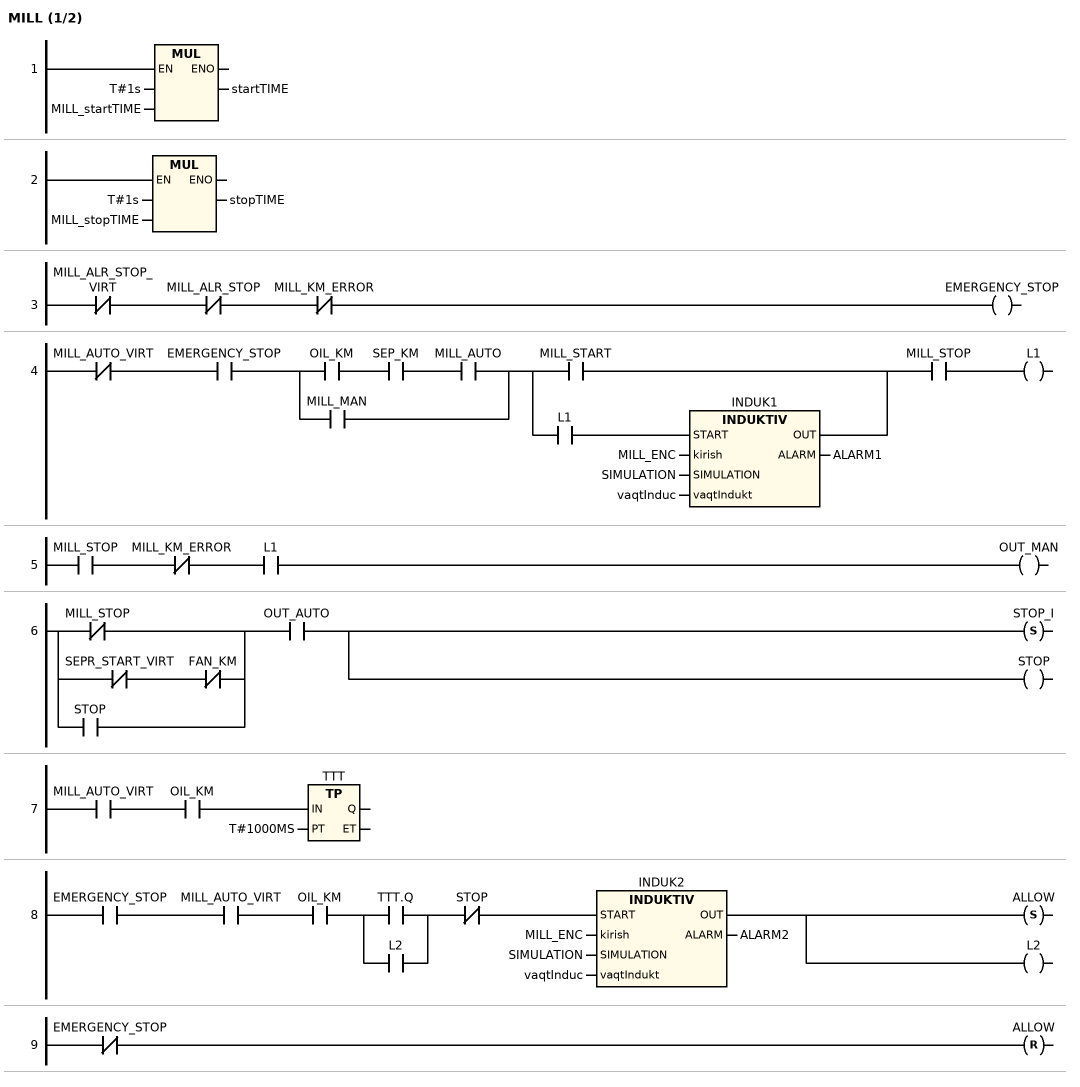
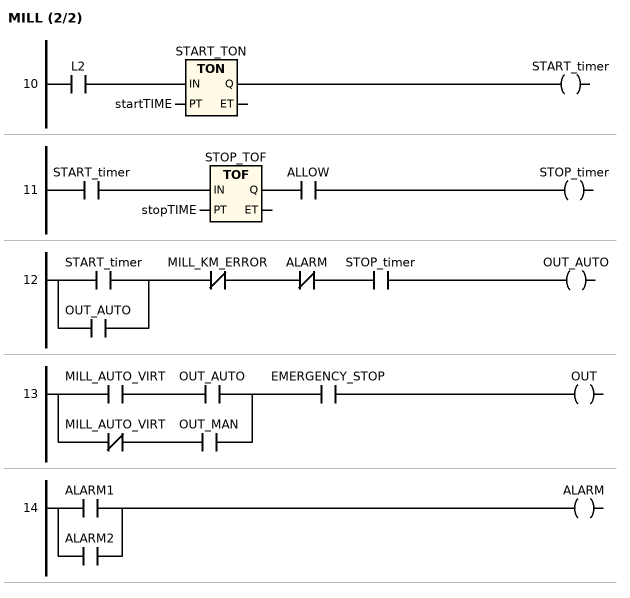
_LD_ (* Ladder Diagram *)
NETWORK 1
	*
		EN --- MUL(T#1s, MILL_startTIME) => startTIME
NETWORK 2
	*
		EN --- MUL(T#1s, MILL_stopTIME) => stopTIME
NETWORK 3
	[/MILL_ALR_STOP_VIRT] - [/MILL_ALR_STOP] - [/MILL_KM_ERROR] --- (EMERGENCY_STOP)
NETWORK 4
	[/MILL_AUTO_VIRT] - [EMERGENCY_STOP] - { [OIL_KM] - [SEP_KM] - [MILL_AUTO] | [MILL_MAN] } - { [MILL_START] | [L1] - INDUK1:INDUKTIV(START: *, kirish: MILL_ENC, SIMULATION: SIMULATION, vaqtIndukt: vaqtInduc, ALARM => ALARM1) } - [MILL_STOP] --- (L1)
NETWORK 5
	[MILL_STOP] - [/MILL_KM_ERROR] - [L1] --- (OUT_MAN)
NETWORK 6
	{ [/MILL_STOP] | [/SEPR_START_VIRT] - [/FAN_KM] | [STOP] } - [OUT_AUTO] --- (S STOP_I) (STOP)
NETWORK 7
	[MILL_AUTO_VIRT] - [OIL_KM] - TTT:TP(IN: *, PT: T#1000MS)
NETWORK 8
	[EMERGENCY_STOP] - [MILL_AUTO_VIRT] - [OIL_KM] - { [TTT.Q] | [L2] } - [/STOP] - INDUK2:INDUKTIV(START: *, kirish: MILL_ENC, SIMULATION: SIMULATION, vaqtIndukt: vaqtInduc, ALARM => ALARM2) --- (S ALLOW) (L2)
NETWORK 9
	[/EMERGENCY_STOP] --- (R ALLOW)
NETWORK 10
	[L2] - START_TON:TON(IN: *, PT: startTIME) --- (START_timer)
NETWORK 11
	[START_timer] - STOP_TOF:TOF(IN: *, PT: stopTIME) - [ALLOW] --- (STOP_timer)
NETWORK 12
	{ [START_timer] | [OUT_AUTO] } - [/MILL_KM_ERROR] - [/ALARM] - [STOP_timer] --- (OUT_AUTO)
NETWORK 13
	{ [MILL_AUTO_VIRT] - [OUT_AUTO] | [/MILL_AUTO_VIRT] - [OUT_MAN] } - [EMERGENCY_STOP] --- (OUT)
NETWORK 14
	{ [ALARM1] | [ALARM2] } --- (ALARM)
_END_LD_
(* the same logic as Structured Text *)
(* Network 1 *)
startTIME := T#1s * MILL_startTIME;
(* Network 2 *)
stopTIME := T#1s * MILL_stopTIME;
(* Network 3 *)
EMERGENCY_STOP := NOT MILL_ALR_STOP_VIRT AND NOT MILL_ALR_STOP AND NOT MILL_KM_ERROR;
(* Network 4 *)
_p1 := NOT MILL_AUTO_VIRT AND EMERGENCY_STOP AND (OIL_KM AND SEP_KM AND MILL_AUTO OR MILL_MAN);
INDUK1(START := _p1 AND L1, kirish := MILL_ENC, SIMULATION := SIMULATION, vaqtIndukt := vaqtInduc);
ALARM1 := INDUK1.ALARM;
L1 := (_p1 AND MILL_START OR INDUK1.OUT) AND MILL_STOP;
(* Network 5 *)
OUT_MAN := MILL_STOP AND NOT MILL_KM_ERROR AND L1;
(* Network 6 *)
_p2 := (NOT MILL_STOP OR NOT SEPR_START_VIRT AND NOT FAN_KM OR STOP) AND OUT_AUTO;
IF _p2 THEN STOP_I := TRUE; END_IF;
STOP := _p2;
(* Network 7 *)
TTT(IN := MILL_AUTO_VIRT AND OIL_KM, PT := T#1000MS);
(* Network 8 *)
INDUK2(START := EMERGENCY_STOP AND MILL_AUTO_VIRT AND OIL_KM AND (TTT.Q OR L2) AND NOT STOP, kirish := MILL_ENC, SIMULATION := SIMULATION, vaqtIndukt := vaqtInduc);
ALARM2 := INDUK2.ALARM;
IF INDUK2.OUT THEN ALLOW := TRUE; END_IF;
L2 := INDUK2.OUT;
(* Network 9 *)
IF NOT EMERGENCY_STOP THEN ALLOW := FALSE; END_IF;
(* Network 10 *)
START_TON(IN := L2, PT := startTIME);
START_timer := START_TON.Q;
(* Network 11 *)
STOP_TOF(IN := START_timer, PT := stopTIME);
STOP_timer := STOP_TOF.Q AND ALLOW;
(* Network 12 *)
OUT_AUTO := (START_timer OR OUT_AUTO) AND NOT MILL_KM_ERROR AND NOT ALARM AND STOP_timer;
(* Network 13 *)
OUT := (MILL_AUTO_VIRT AND OUT_AUTO OR NOT MILL_AUTO_VIRT AND OUT_MAN) AND EMERGENCY_STOP;
(* Network 14 *)
ALARM := ALARM1 OR ALARM2;
END_FUNCTION_BLOCK

(* POU FAN, LD *)
FUNCTION_BLOCK FAN
VAR_INPUT
	EN : BOOL;
	MILL_ALR_STOP: BOOL;
	MILL_ALR_STOP_VIRT : BOOL;
	MILL_AUTO : BOOL;
	MILL_AUTO_VIRT : BOOL;
	MILL_MAN : BOOL;
	FAN_START : BOOL;
	VIBRATOR_T : BOOL;

	FAN_STOP : BOOL;
	MILL_KM : BOOL;

	FAN_KM_ERROR : BOOL;
	SEPR_START_VIRT : BOOL;
	FAN_startTIME : WORD;
	FAN_stopTIME : WORD;
END_VAR

VAR_OUTPUT
	OUT : BOOL;
	ALARM : BOOL;
END_VAR
VAR
	INDUK1: INDUKTIV;
	INDUK2: INDUKTIV;
	OUT_MAN: BOOL;
	OUT_AUTO: BOOL;
	START_TON : TON;
	STOP_TOF : TOF;
	startTIME : TIME;
	stopTIME : TIME;
	L1: BOOL;
	L2: BOOL;
	ES: BOOL;
	EMERGENCY_STOP: BOOL;
	ALARM1 : BOOL;
	ALARM2 : BOOL;

	STOP: BOOL;
	ALLOW: BOOL;
	START_timer: BOOL;
	STOP_timer: BOOL;
	TTT : TP;
END_VAR
VAR (* helpers for the ST form of the networks *)
	_p1 : BOOL;
END_VAR
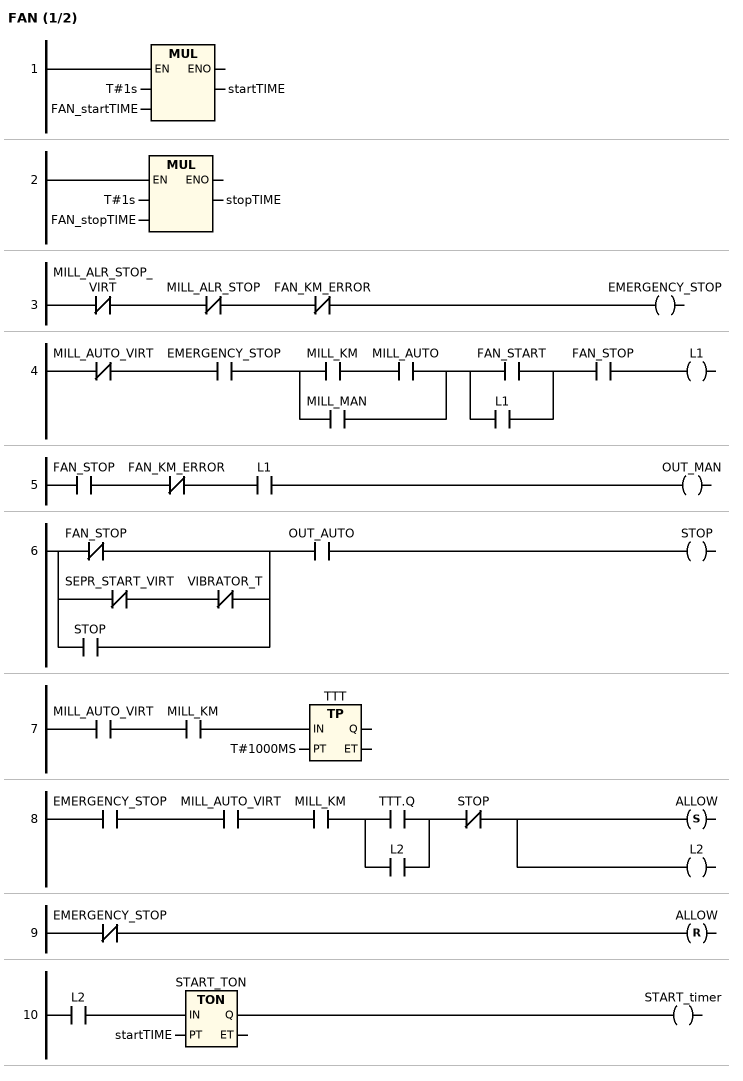
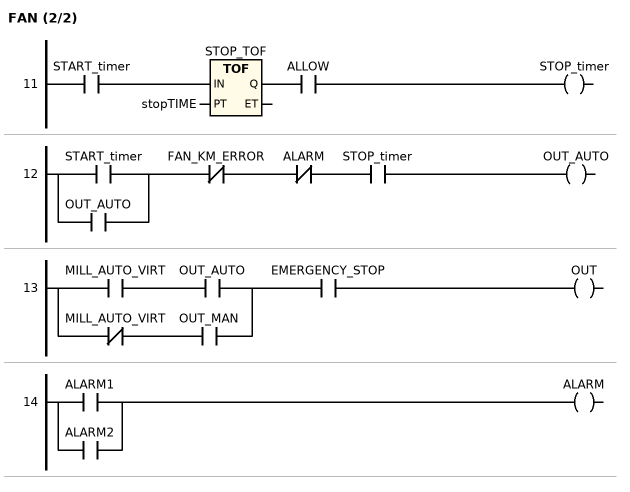
_LD_ (* Ladder Diagram *)
NETWORK 1
	*
		EN --- MUL(T#1s, FAN_startTIME) => startTIME
NETWORK 2
	*
		EN --- MUL(T#1s, FAN_stopTIME) => stopTIME
NETWORK 3
	[/MILL_ALR_STOP_VIRT] - [/MILL_ALR_STOP] - [/FAN_KM_ERROR] --- (EMERGENCY_STOP)
NETWORK 4
	[/MILL_AUTO_VIRT] - [EMERGENCY_STOP] - { [MILL_KM] - [MILL_AUTO] | [MILL_MAN] } - { [FAN_START] | [L1] } - [FAN_STOP] --- (L1)
NETWORK 5
	[FAN_STOP] - [/FAN_KM_ERROR] - [L1] --- (OUT_MAN)
NETWORK 6
	{ [/FAN_STOP] | [/SEPR_START_VIRT] - [/VIBRATOR_T] | [STOP] } - [OUT_AUTO] --- (STOP)
NETWORK 7
	[MILL_AUTO_VIRT] - [MILL_KM] - TTT:TP(IN: *, PT: T#1000MS)
NETWORK 8
	[EMERGENCY_STOP] - [MILL_AUTO_VIRT] - [MILL_KM] - { [TTT.Q] | [L2] } - [/STOP] --- (S ALLOW) (L2)
NETWORK 9
	[/EMERGENCY_STOP] --- (R ALLOW)
NETWORK 10
	[L2] - START_TON:TON(IN: *, PT: startTIME) --- (START_timer)
NETWORK 11
	[START_timer] - STOP_TOF:TOF(IN: *, PT: stopTIME) - [ALLOW] --- (STOP_timer)
NETWORK 12
	{ [START_timer] | [OUT_AUTO] } - [/FAN_KM_ERROR] - [/ALARM] - [STOP_timer] --- (OUT_AUTO)
NETWORK 13
	{ [MILL_AUTO_VIRT] - [OUT_AUTO] | [/MILL_AUTO_VIRT] - [OUT_MAN] } - [EMERGENCY_STOP] --- (OUT)
NETWORK 14
	{ [ALARM1] | [ALARM2] } --- (ALARM)
_END_LD_
(* the same logic as Structured Text *)
(* Network 1 *)
startTIME := T#1s * FAN_startTIME;
(* Network 2 *)
stopTIME := T#1s * FAN_stopTIME;
(* Network 3 *)
EMERGENCY_STOP := NOT MILL_ALR_STOP_VIRT AND NOT MILL_ALR_STOP AND NOT FAN_KM_ERROR;
(* Network 4 *)
L1 := NOT MILL_AUTO_VIRT AND EMERGENCY_STOP AND (MILL_KM AND MILL_AUTO OR MILL_MAN) AND (FAN_START OR L1) AND FAN_STOP;
(* Network 5 *)
OUT_MAN := FAN_STOP AND NOT FAN_KM_ERROR AND L1;
(* Network 6 *)
STOP := (NOT FAN_STOP OR NOT SEPR_START_VIRT AND NOT VIBRATOR_T OR STOP) AND OUT_AUTO;
(* Network 7 *)
TTT(IN := MILL_AUTO_VIRT AND MILL_KM, PT := T#1000MS);
(* Network 8 *)
_p1 := EMERGENCY_STOP AND MILL_AUTO_VIRT AND MILL_KM AND (TTT.Q OR L2) AND NOT STOP;
IF _p1 THEN ALLOW := TRUE; END_IF;
L2 := _p1;
(* Network 9 *)
IF NOT EMERGENCY_STOP THEN ALLOW := FALSE; END_IF;
(* Network 10 *)
START_TON(IN := L2, PT := startTIME);
START_timer := START_TON.Q;
(* Network 11 *)
STOP_TOF(IN := START_timer, PT := stopTIME);
STOP_timer := STOP_TOF.Q AND ALLOW;
(* Network 12 *)
OUT_AUTO := (START_timer OR OUT_AUTO) AND NOT FAN_KM_ERROR AND NOT ALARM AND STOP_timer;
(* Network 13 *)
OUT := (MILL_AUTO_VIRT AND OUT_AUTO OR NOT MILL_AUTO_VIRT AND OUT_MAN) AND EMERGENCY_STOP;
(* Network 14 *)
ALARM := ALARM1 OR ALARM2;
END_FUNCTION_BLOCK

(* POU CONV, LD *)
FUNCTION_BLOCK CONV
VAR_INPUT
	EN : BOOL;
	MILL_ALR_STOP: BOOL;
	MILL_ALR_STOP_VIRT : BOOL;
	MILL_AUTO : BOOL;
	MILL_AUTO_VIRT : BOOL;
	MILL_MAN : BOOL;
	CONV_START : BOOL;
	FAN_KM : BOOL;
	MILL_KM : BOOL;
	CONV_ENC : BOOL;
	CONV_STOP : BOOL;
	VIBRATOR_T : BOOL;
	CONV_KM_ERROR : BOOL;
	SIMULATION : BOOL := TRUE;
	MATER_FULL : BOOL;
	SEPR_START_VIRT : BOOL;
	vaqtInduc : WORD := 15;
END_VAR

VAR_OUTPUT
	OUT : BOOL;
	ALARM : BOOL;
END_VAR
VAR
	INDUK1: INDUKTIV;
	INDUK2: INDUKTIV;
	OUT_MAN: BOOL;
	OUT_AUTO: BOOL;
	START_TON : TON;
	STOP_TOF : TOF;
	startTIME : TIME;
	stopTIME : TIME;
	L1: BOOL;
	L2: BOOL;
	ES: BOOL;
	EMERGENCY_STOP: BOOL;
	ALARM1 : BOOL;
	ALARM2 : BOOL;

	STOP: BOOL;
	ALLOW: BOOL;
	START_timer: BOOL;
	STOP_timer: BOOL;
	TTT : TP;
END_VAR
VAR (* helpers for the ST form of the networks *)
	_p1 : BOOL;
END_VAR
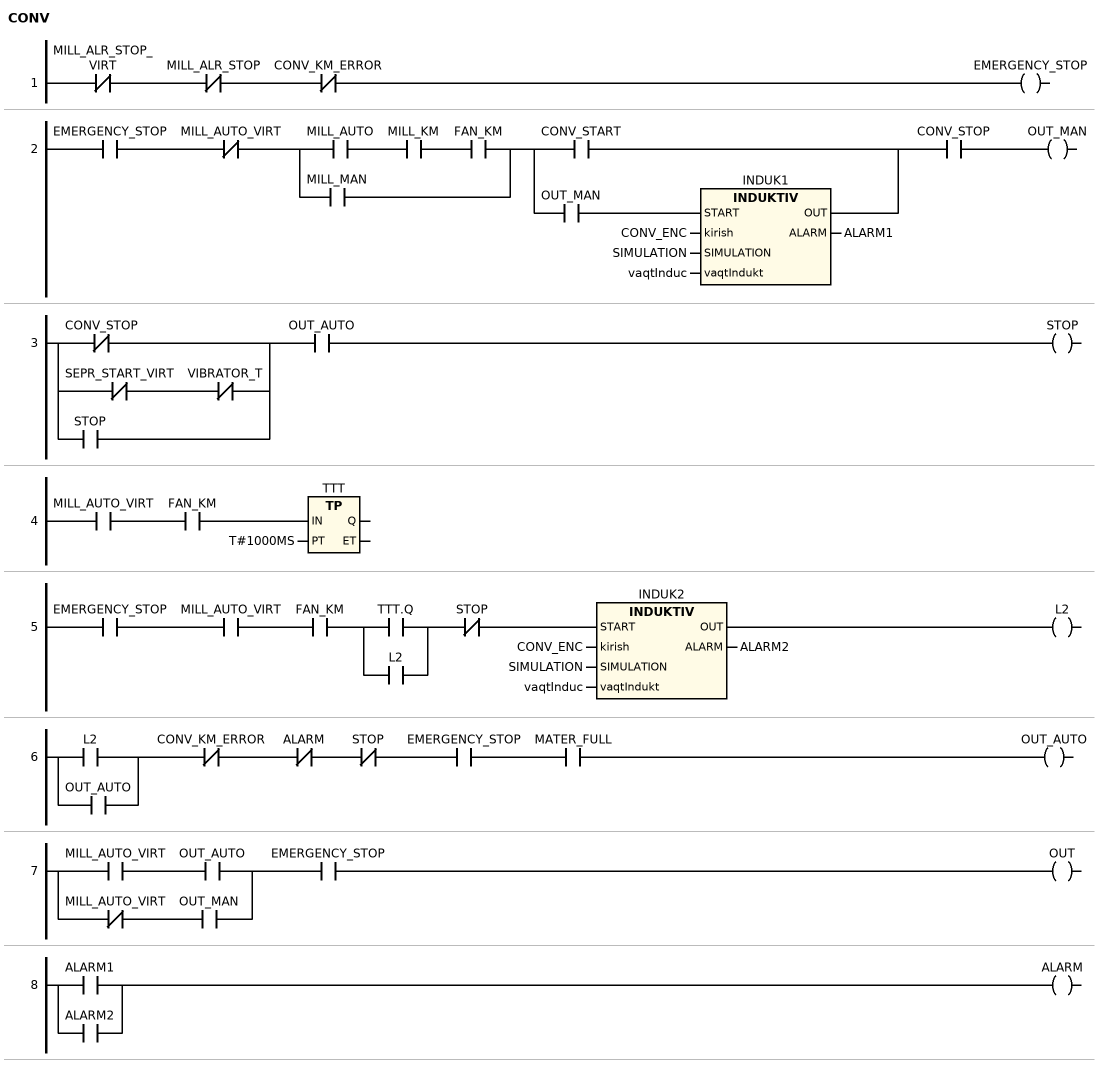
_LD_ (* Ladder Diagram *)
NETWORK 1
	[/MILL_ALR_STOP_VIRT] - [/MILL_ALR_STOP] - [/CONV_KM_ERROR] --- (EMERGENCY_STOP)
NETWORK 2
	[EMERGENCY_STOP] - [/MILL_AUTO_VIRT] - { [MILL_AUTO] - [MILL_KM] - [FAN_KM] | [MILL_MAN] } - { [CONV_START] | [OUT_MAN] - INDUK1:INDUKTIV(START: *, kirish: CONV_ENC, SIMULATION: SIMULATION, vaqtIndukt: vaqtInduc, ALARM => ALARM1) } - [CONV_STOP] --- (OUT_MAN)
NETWORK 3
	{ [/CONV_STOP] | [/SEPR_START_VIRT] - [/VIBRATOR_T] | [STOP] } - [OUT_AUTO] --- (STOP)
NETWORK 4
	[MILL_AUTO_VIRT] - [FAN_KM] - TTT:TP(IN: *, PT: T#1000MS)
NETWORK 5
	[EMERGENCY_STOP] - [MILL_AUTO_VIRT] - [FAN_KM] - { [TTT.Q] | [L2] } - [/STOP] - INDUK2:INDUKTIV(START: *, kirish: CONV_ENC, SIMULATION: SIMULATION, vaqtIndukt: vaqtInduc, ALARM => ALARM2) --- (L2)
NETWORK 6
	{ [L2] | [OUT_AUTO] } - [/CONV_KM_ERROR] - [/ALARM] - [/STOP] - [EMERGENCY_STOP] - [MATER_FULL] --- (OUT_AUTO)
NETWORK 7
	{ [MILL_AUTO_VIRT] - [OUT_AUTO] | [/MILL_AUTO_VIRT] - [OUT_MAN] } - [EMERGENCY_STOP] --- (OUT)
NETWORK 8
	{ [ALARM1] | [ALARM2] } --- (ALARM)
_END_LD_
(* the same logic as Structured Text *)
(* Network 1 *)
EMERGENCY_STOP := NOT MILL_ALR_STOP_VIRT AND NOT MILL_ALR_STOP AND NOT CONV_KM_ERROR;
(* Network 2 *)
_p1 := EMERGENCY_STOP AND NOT MILL_AUTO_VIRT AND (MILL_AUTO AND MILL_KM AND FAN_KM OR MILL_MAN);
INDUK1(START := _p1 AND OUT_MAN, kirish := CONV_ENC, SIMULATION := SIMULATION, vaqtIndukt := vaqtInduc);
ALARM1 := INDUK1.ALARM;
OUT_MAN := (_p1 AND CONV_START OR INDUK1.OUT) AND CONV_STOP;
(* Network 3 *)
STOP := (NOT CONV_STOP OR NOT SEPR_START_VIRT AND NOT VIBRATOR_T OR STOP) AND OUT_AUTO;
(* Network 4 *)
TTT(IN := MILL_AUTO_VIRT AND FAN_KM, PT := T#1000MS);
(* Network 5 *)
INDUK2(START := EMERGENCY_STOP AND MILL_AUTO_VIRT AND FAN_KM AND (TTT.Q OR L2) AND NOT STOP, kirish := CONV_ENC, SIMULATION := SIMULATION, vaqtIndukt := vaqtInduc);
ALARM2 := INDUK2.ALARM;
L2 := INDUK2.OUT;
(* Network 6 *)
OUT_AUTO := (L2 OR OUT_AUTO) AND NOT CONV_KM_ERROR AND NOT ALARM AND NOT STOP AND EMERGENCY_STOP AND MATER_FULL;
(* Network 7 *)
OUT := (MILL_AUTO_VIRT AND OUT_AUTO OR NOT MILL_AUTO_VIRT AND OUT_MAN) AND EMERGENCY_STOP;
(* Network 8 *)
ALARM := ALARM1 OR ALARM2;
END_FUNCTION_BLOCK

(* POU ALARMS, LD *)
PROGRAM ALARMS
VAR
	tofELV: TON;
	tofSHNK3: TON;
	tofSHNK4: TON;
	tofSHNK_SKL_3: TON;
	tofSHNK_SKL_4: TON;
	tofSTAR_31: TON;
	tofSTAR_32: TON;
	tofSTAR_41: TON;
	tofSTAR_42: TON;
	tofSEPR_3: TON;
	tofSEPR_4: TON;
	tofOIL_3: TON;
	tofOIL_4: TON;
	tofMILL_3: TON;
	tofMILL_4: TON;
	tofFAN_3: TON;
	tofFAN_4: TON;
	tofCONV_3: TON;
	tofCONV_4: TON;
	tofVIB_3: TON;
	tofVIB_4: TON;

	vaqt : TIME := T#30S;
END_VAR
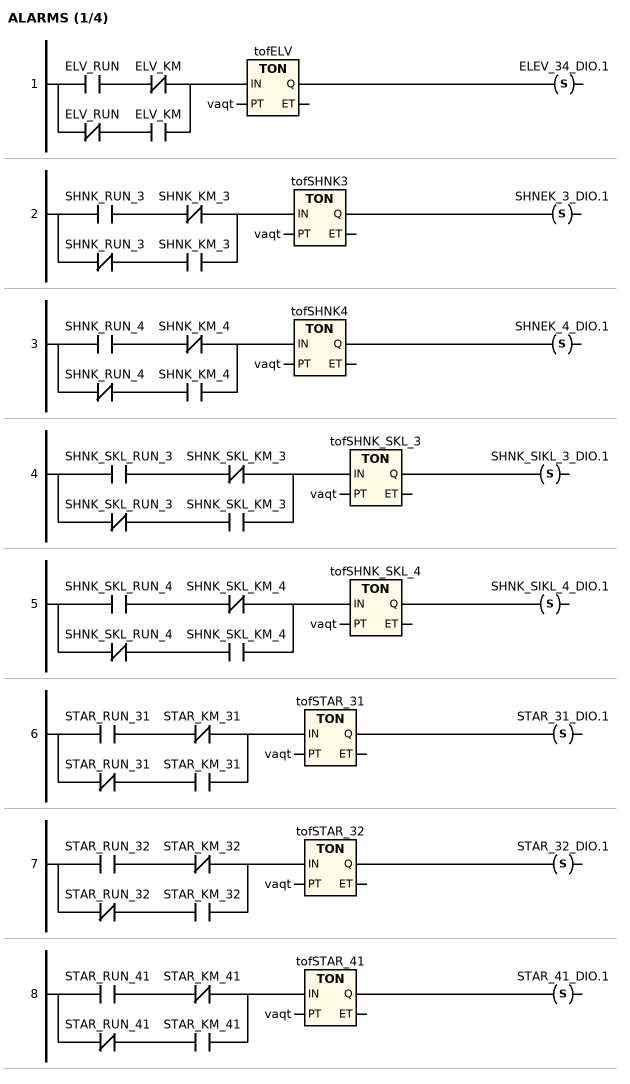
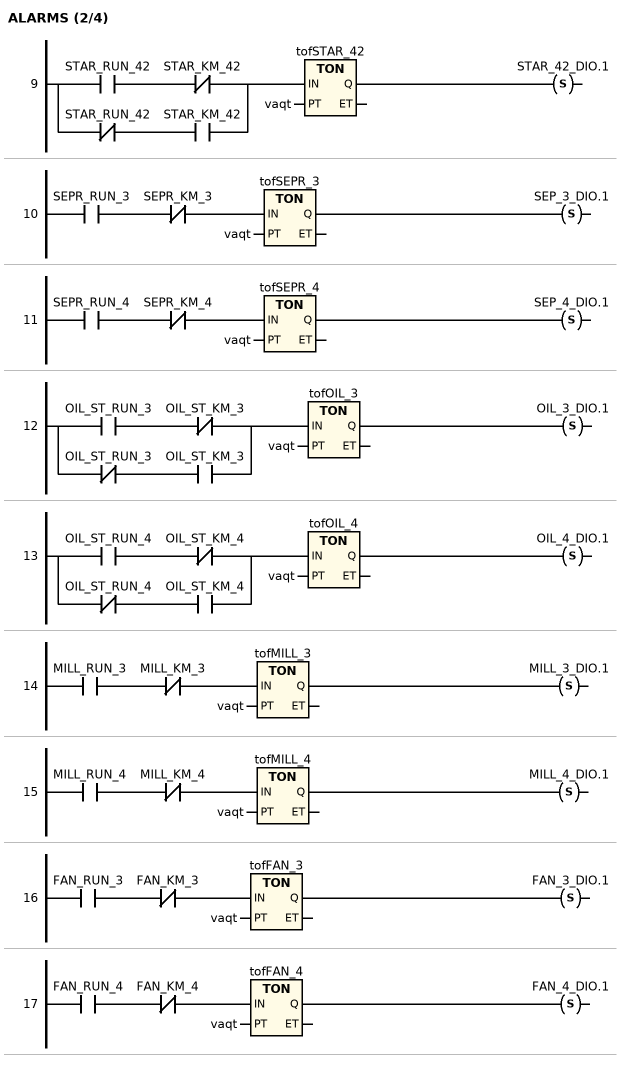
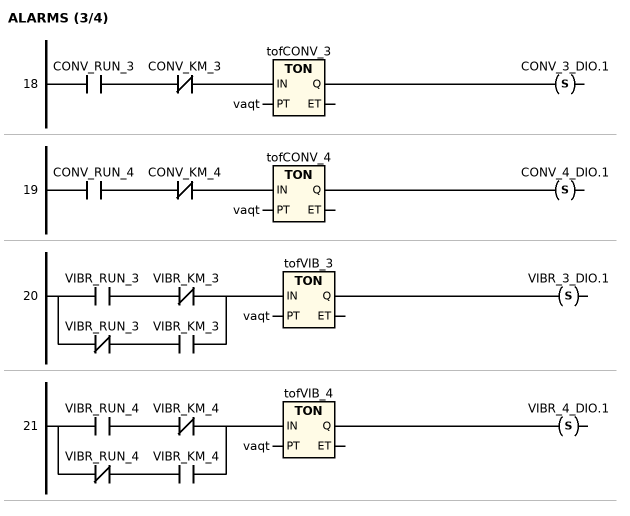
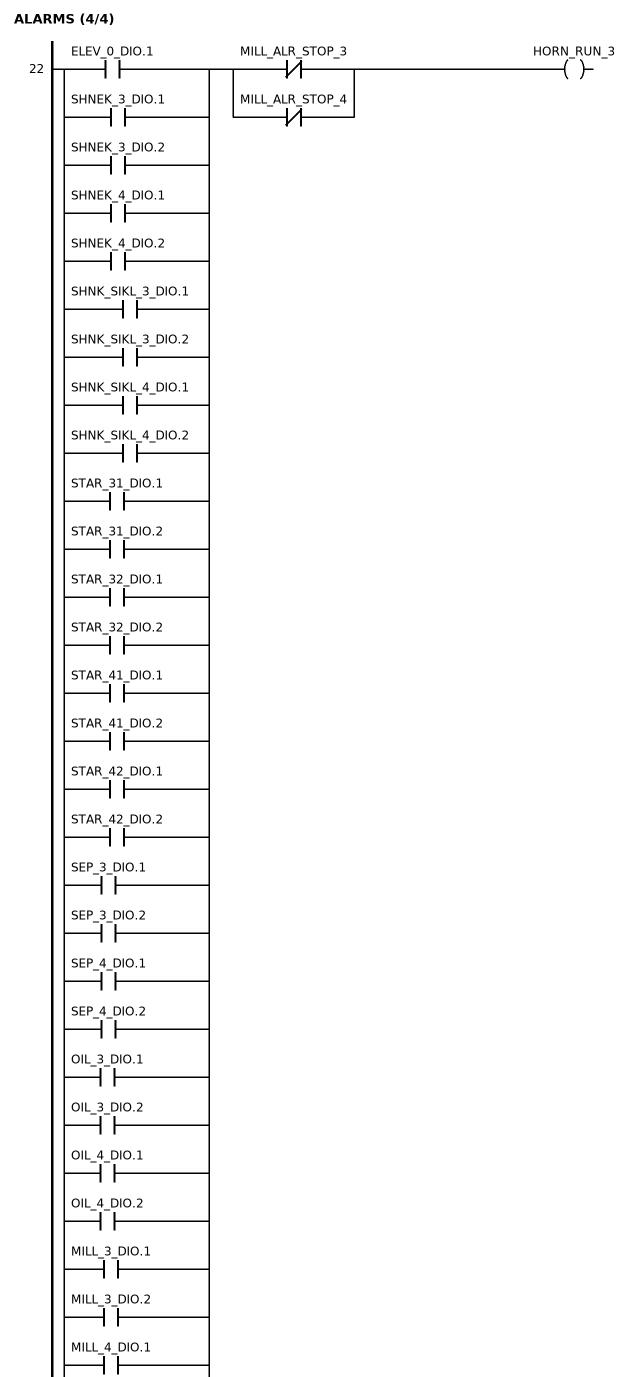
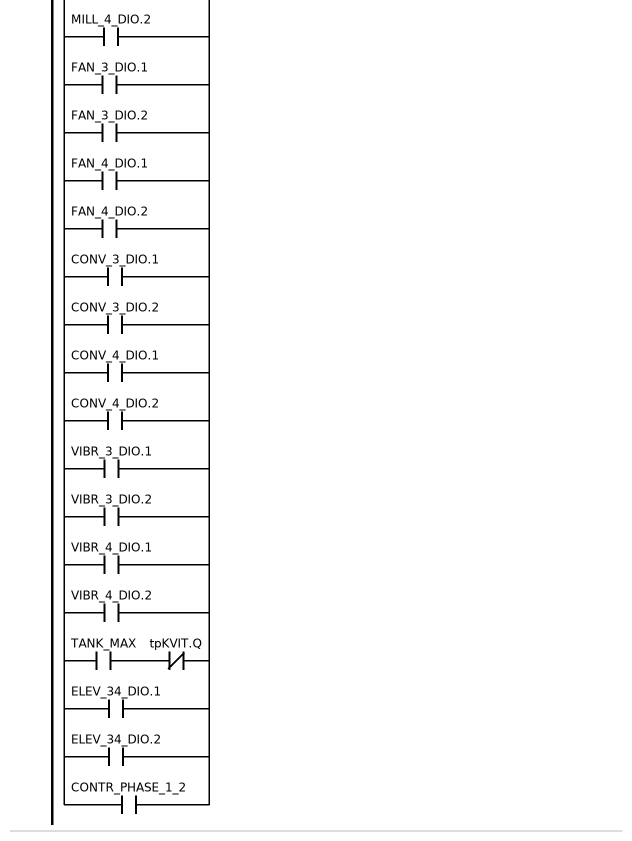
_LD_ (* Ladder Diagram *)
NETWORK 1
	{ [ELV_RUN] - [/ELV_KM] | [/ELV_RUN] - [ELV_KM] } - tofELV:TON(IN: *, PT: vaqt) --- (S ELEV_34_DIO.1)
NETWORK 2
	{ [SHNK_RUN_3] - [/SHNK_KM_3] | [/SHNK_RUN_3] - [SHNK_KM_3] } - tofSHNK3:TON(IN: *, PT: vaqt) --- (S SHNEK_3_DIO.1)
NETWORK 3
	{ [SHNK_RUN_4] - [/SHNK_KM_4] | [/SHNK_RUN_4] - [SHNK_KM_4] } - tofSHNK4:TON(IN: *, PT: vaqt) --- (S SHNEK_4_DIO.1)
NETWORK 4
	{ [SHNK_SKL_RUN_3] - [/SHNK_SKL_KM_3] | [/SHNK_SKL_RUN_3] - [SHNK_SKL_KM_3] } - tofSHNK_SKL_3:TON(IN: *, PT: vaqt) --- (S SHNK_SIKL_3_DIO.1)
NETWORK 5
	{ [SHNK_SKL_RUN_4] - [/SHNK_SKL_KM_4] | [/SHNK_SKL_RUN_4] - [SHNK_SKL_KM_4] } - tofSHNK_SKL_4:TON(IN: *, PT: vaqt) --- (S SHNK_SIKL_4_DIO.1)
NETWORK 6
	{ [STAR_RUN_31] - [/STAR_KM_31] | [/STAR_RUN_31] - [STAR_KM_31] } - tofSTAR_31:TON(IN: *, PT: vaqt) --- (S STAR_31_DIO.1)
NETWORK 7
	{ [STAR_RUN_32] - [/STAR_KM_32] | [/STAR_RUN_32] - [STAR_KM_32] } - tofSTAR_32:TON(IN: *, PT: vaqt) --- (S STAR_32_DIO.1)
NETWORK 8
	{ [STAR_RUN_41] - [/STAR_KM_41] | [/STAR_RUN_41] - [STAR_KM_41] } - tofSTAR_41:TON(IN: *, PT: vaqt) --- (S STAR_41_DIO.1)
NETWORK 9
	{ [STAR_RUN_42] - [/STAR_KM_42] | [/STAR_RUN_42] - [STAR_KM_42] } - tofSTAR_42:TON(IN: *, PT: vaqt) --- (S STAR_42_DIO.1)
NETWORK 10
	[SEPR_RUN_3] - [/SEPR_KM_3] - tofSEPR_3:TON(IN: *, PT: vaqt) --- (S SEP_3_DIO.1)
NETWORK 11
	[SEPR_RUN_4] - [/SEPR_KM_4] - tofSEPR_4:TON(IN: *, PT: vaqt) --- (S SEP_4_DIO.1)
NETWORK 12
	{ [OIL_ST_RUN_3] - [/OIL_ST_KM_3] | [/OIL_ST_RUN_3] - [OIL_ST_KM_3] } - tofOIL_3:TON(IN: *, PT: vaqt) --- (S OIL_3_DIO.1)
NETWORK 13
	{ [OIL_ST_RUN_4] - [/OIL_ST_KM_4] | [/OIL_ST_RUN_4] - [OIL_ST_KM_4] } - tofOIL_4:TON(IN: *, PT: vaqt) --- (S OIL_4_DIO.1)
NETWORK 14
	[MILL_RUN_3] - [/MILL_KM_3] - tofMILL_3:TON(IN: *, PT: vaqt) --- (S MILL_3_DIO.1)
NETWORK 15
	[MILL_RUN_4] - [/MILL_KM_4] - tofMILL_4:TON(IN: *, PT: vaqt) --- (S MILL_4_DIO.1)
NETWORK 16
	[FAN_RUN_3] - [/FAN_KM_3] - tofFAN_3:TON(IN: *, PT: vaqt) --- (S FAN_3_DIO.1)
NETWORK 17
	[FAN_RUN_4] - [/FAN_KM_4] - tofFAN_4:TON(IN: *, PT: vaqt) --- (S FAN_4_DIO.1)
NETWORK 18
	[CONV_RUN_3] - [/CONV_KM_3] - tofCONV_3:TON(IN: *, PT: vaqt) --- (S CONV_3_DIO.1)
NETWORK 19
	[CONV_RUN_4] - [/CONV_KM_4] - tofCONV_4:TON(IN: *, PT: vaqt) --- (S CONV_4_DIO.1)
NETWORK 20
	{ [VIBR_RUN_3] - [/VIBR_KM_3] | [/VIBR_RUN_3] - [VIBR_KM_3] } - tofVIB_3:TON(IN: *, PT: vaqt) --- (S VIBR_3_DIO.1)
NETWORK 21
	{ [VIBR_RUN_4] - [/VIBR_KM_4] | [/VIBR_RUN_4] - [VIBR_KM_4] } - tofVIB_4:TON(IN: *, PT: vaqt) --- (S VIBR_4_DIO.1)
NETWORK 22
	{ [ELEV_0_DIO.1] | [SHNEK_3_DIO.1] | [SHNEK_3_DIO.2] | [SHNEK_4_DIO.1] | [SHNEK_4_DIO.2] | [SHNK_SIKL_3_DIO.1] | [SHNK_SIKL_3_DIO.2] | [SHNK_SIKL_4_DIO.1] | [SHNK_SIKL_4_DIO.2] | [STAR_31_DIO.1] | [STAR_31_DIO.2] | [STAR_32_DIO.1] | [STAR_32_DIO.2] | [STAR_41_DIO.1] | [STAR_41_DIO.2] | [STAR_42_DIO.1] | [STAR_42_DIO.2] | [SEP_3_DIO.1] | [SEP_3_DIO.2] | [SEP_4_DIO.1] | [SEP_4_DIO.2] | [OIL_3_DIO.1] | [OIL_3_DIO.2] | [OIL_4_DIO.1] | [OIL_4_DIO.2] | [MILL_3_DIO.1] | [MILL_3_DIO.2] | [MILL_4_DIO.1] | [MILL_4_DIO.2] | [FAN_3_DIO.1] | [FAN_3_DIO.2] | [FAN_4_DIO.1] | [FAN_4_DIO.2] | [CONV_3_DIO.1] | [CONV_3_DIO.2] | [CONV_4_DIO.1] | [CONV_4_DIO.2] | [VIBR_3_DIO.1] | [VIBR_3_DIO.2] | [VIBR_4_DIO.1] | [VIBR_4_DIO.2] | [TANK_MAX] - [/tpKVIT.Q] | [ELEV_34_DIO.1] | [ELEV_34_DIO.2] | [CONTR_PHASE_1_2] } - { [/MILL_ALR_STOP_3] | [/MILL_ALR_STOP_4] } --- (HORN_RUN_3)
_END_LD_
(* the same logic as Structured Text *)
(* Network 1 *)
tofELV(IN := ELV_RUN AND NOT ELV_KM OR NOT ELV_RUN AND ELV_KM, PT := vaqt);
IF tofELV.Q THEN ELEV_34_DIO.1 := TRUE; END_IF;
(* Network 2 *)
tofSHNK3(IN := SHNK_RUN_3 AND NOT SHNK_KM_3 OR NOT SHNK_RUN_3 AND SHNK_KM_3, PT := vaqt);
IF tofSHNK3.Q THEN SHNEK_3_DIO.1 := TRUE; END_IF;
(* Network 3 *)
tofSHNK4(IN := SHNK_RUN_4 AND NOT SHNK_KM_4 OR NOT SHNK_RUN_4 AND SHNK_KM_4, PT := vaqt);
IF tofSHNK4.Q THEN SHNEK_4_DIO.1 := TRUE; END_IF;
(* Network 4 *)
tofSHNK_SKL_3(IN := SHNK_SKL_RUN_3 AND NOT SHNK_SKL_KM_3 OR NOT SHNK_SKL_RUN_3 AND SHNK_SKL_KM_3, PT := vaqt);
IF tofSHNK_SKL_3.Q THEN SHNK_SIKL_3_DIO.1 := TRUE; END_IF;
(* Network 5 *)
tofSHNK_SKL_4(IN := SHNK_SKL_RUN_4 AND NOT SHNK_SKL_KM_4 OR NOT SHNK_SKL_RUN_4 AND SHNK_SKL_KM_4, PT := vaqt);
IF tofSHNK_SKL_4.Q THEN SHNK_SIKL_4_DIO.1 := TRUE; END_IF;
(* Network 6 *)
tofSTAR_31(IN := STAR_RUN_31 AND NOT STAR_KM_31 OR NOT STAR_RUN_31 AND STAR_KM_31, PT := vaqt);
IF tofSTAR_31.Q THEN STAR_31_DIO.1 := TRUE; END_IF;
(* Network 7 *)
tofSTAR_32(IN := STAR_RUN_32 AND NOT STAR_KM_32 OR NOT STAR_RUN_32 AND STAR_KM_32, PT := vaqt);
IF tofSTAR_32.Q THEN STAR_32_DIO.1 := TRUE; END_IF;
(* Network 8 *)
tofSTAR_41(IN := STAR_RUN_41 AND NOT STAR_KM_41 OR NOT STAR_RUN_41 AND STAR_KM_41, PT := vaqt);
IF tofSTAR_41.Q THEN STAR_41_DIO.1 := TRUE; END_IF;
(* Network 9 *)
tofSTAR_42(IN := STAR_RUN_42 AND NOT STAR_KM_42 OR NOT STAR_RUN_42 AND STAR_KM_42, PT := vaqt);
IF tofSTAR_42.Q THEN STAR_42_DIO.1 := TRUE; END_IF;
(* Network 10 *)
tofSEPR_3(IN := SEPR_RUN_3 AND NOT SEPR_KM_3, PT := vaqt);
IF tofSEPR_3.Q THEN SEP_3_DIO.1 := TRUE; END_IF;
(* Network 11 *)
tofSEPR_4(IN := SEPR_RUN_4 AND NOT SEPR_KM_4, PT := vaqt);
IF tofSEPR_4.Q THEN SEP_4_DIO.1 := TRUE; END_IF;
(* Network 12 *)
tofOIL_3(IN := OIL_ST_RUN_3 AND NOT OIL_ST_KM_3 OR NOT OIL_ST_RUN_3 AND OIL_ST_KM_3, PT := vaqt);
IF tofOIL_3.Q THEN OIL_3_DIO.1 := TRUE; END_IF;
(* Network 13 *)
tofOIL_4(IN := OIL_ST_RUN_4 AND NOT OIL_ST_KM_4 OR NOT OIL_ST_RUN_4 AND OIL_ST_KM_4, PT := vaqt);
IF tofOIL_4.Q THEN OIL_4_DIO.1 := TRUE; END_IF;
(* Network 14 *)
tofMILL_3(IN := MILL_RUN_3 AND NOT MILL_KM_3, PT := vaqt);
IF tofMILL_3.Q THEN MILL_3_DIO.1 := TRUE; END_IF;
(* Network 15 *)
tofMILL_4(IN := MILL_RUN_4 AND NOT MILL_KM_4, PT := vaqt);
IF tofMILL_4.Q THEN MILL_4_DIO.1 := TRUE; END_IF;
(* Network 16 *)
tofFAN_3(IN := FAN_RUN_3 AND NOT FAN_KM_3, PT := vaqt);
IF tofFAN_3.Q THEN FAN_3_DIO.1 := TRUE; END_IF;
(* Network 17 *)
tofFAN_4(IN := FAN_RUN_4 AND NOT FAN_KM_4, PT := vaqt);
IF tofFAN_4.Q THEN FAN_4_DIO.1 := TRUE; END_IF;
(* Network 18 *)
tofCONV_3(IN := CONV_RUN_3 AND NOT CONV_KM_3, PT := vaqt);
IF tofCONV_3.Q THEN CONV_3_DIO.1 := TRUE; END_IF;
(* Network 19 *)
tofCONV_4(IN := CONV_RUN_4 AND NOT CONV_KM_4, PT := vaqt);
IF tofCONV_4.Q THEN CONV_4_DIO.1 := TRUE; END_IF;
(* Network 20 *)
tofVIB_3(IN := VIBR_RUN_3 AND NOT VIBR_KM_3 OR NOT VIBR_RUN_3 AND VIBR_KM_3, PT := vaqt);
IF tofVIB_3.Q THEN VIBR_3_DIO.1 := TRUE; END_IF;
(* Network 21 *)
tofVIB_4(IN := VIBR_RUN_4 AND NOT VIBR_KM_4 OR NOT VIBR_RUN_4 AND VIBR_KM_4, PT := vaqt);
IF tofVIB_4.Q THEN VIBR_4_DIO.1 := TRUE; END_IF;
(* Network 22 *)
HORN_RUN_3 := (ELEV_0_DIO.1 OR SHNEK_3_DIO.1 OR SHNEK_3_DIO.2 OR SHNEK_4_DIO.1 OR SHNEK_4_DIO.2 OR SHNK_SIKL_3_DIO.1 OR SHNK_SIKL_3_DIO.2 OR SHNK_SIKL_4_DIO.1 OR SHNK_SIKL_4_DIO.2 OR STAR_31_DIO.1 OR STAR_31_DIO.2 OR STAR_32_DIO.1 OR STAR_32_DIO.2 OR STAR_41_DIO.1 OR STAR_41_DIO.2 OR STAR_42_DIO.1 OR STAR_42_DIO.2 OR SEP_3_DIO.1 OR SEP_3_DIO.2 OR SEP_4_DIO.1 OR SEP_4_DIO.2 OR OIL_3_DIO.1 OR OIL_3_DIO.2 OR OIL_4_DIO.1 OR OIL_4_DIO.2 OR MILL_3_DIO.1 OR MILL_3_DIO.2 OR MILL_4_DIO.1 OR MILL_4_DIO.2 OR FAN_3_DIO.1 OR FAN_3_DIO.2 OR FAN_4_DIO.1 OR FAN_4_DIO.2 OR CONV_3_DIO.1 OR CONV_3_DIO.2 OR CONV_4_DIO.1 OR CONV_4_DIO.2 OR VIBR_3_DIO.1 OR VIBR_3_DIO.2 OR VIBR_4_DIO.1 OR VIBR_4_DIO.2 OR TANK_MAX AND NOT tpKVIT.Q OR ELEV_34_DIO.1 OR ELEV_34_DIO.2 OR CONTR_PHASE_1_2) AND (NOT MILL_ALR_STOP_3 OR NOT MILL_ALR_STOP_4);
END_PROGRAM

(* POU RESET_ALRM, LD *)
PROGRAM RESET_ALRM
VAR
END_VAR
VAR (* helpers for the ST form of the networks *)
	_p1 : BOOL;
END_VAR
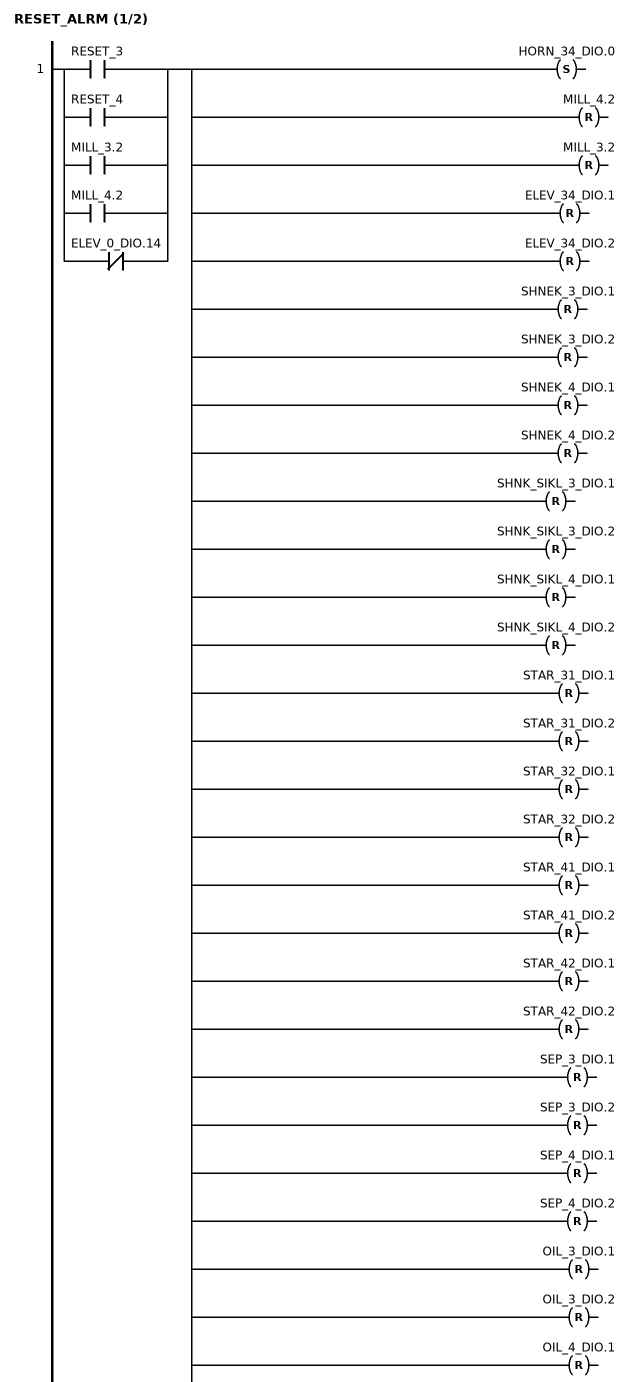
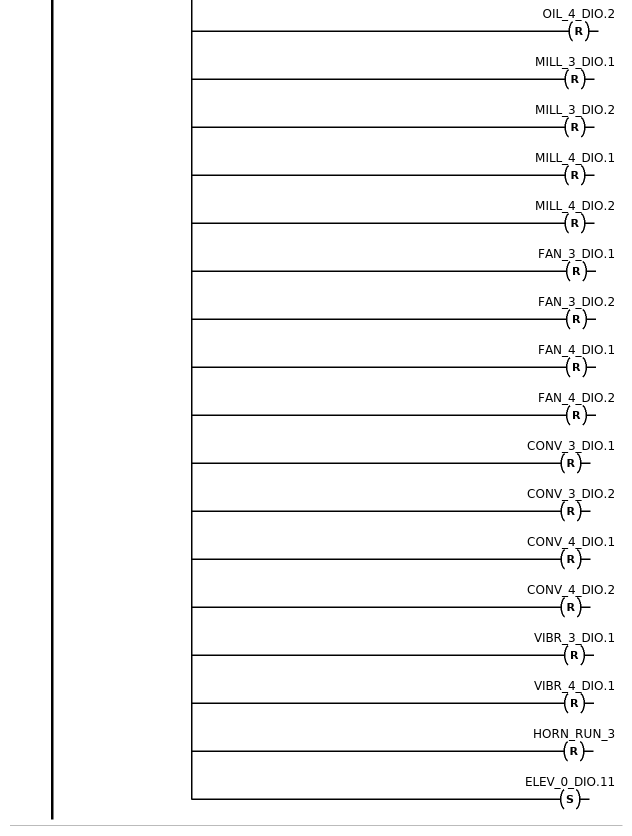
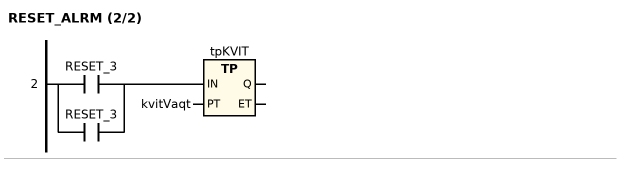
_LD_ (* Ladder Diagram *)
NETWORK 1
	{ [RESET_3] | [RESET_4] | [MILL_3.2] | [MILL_4.2] | [/ELEV_0_DIO.14] } --- (S HORN_34_DIO.0) (R MILL_4.2) (R MILL_3.2) (R ELEV_34_DIO.1) (R ELEV_34_DIO.2) (R SHNEK_3_DIO.1) (R SHNEK_3_DIO.2) (R SHNEK_4_DIO.1) (R SHNEK_4_DIO.2) (R SHNK_SIKL_3_DIO.1) (R SHNK_SIKL_3_DIO.2) (R SHNK_SIKL_4_DIO.1) (R SHNK_SIKL_4_DIO.2) (R STAR_31_DIO.1) (R STAR_31_DIO.2) (R STAR_32_DIO.1) (R STAR_32_DIO.2) (R STAR_41_DIO.1) (R STAR_41_DIO.2) (R STAR_42_DIO.1) (R STAR_42_DIO.2) (R SEP_3_DIO.1) (R SEP_3_DIO.2) (R SEP_4_DIO.1) (R SEP_4_DIO.2) (R OIL_3_DIO.1) (R OIL_3_DIO.2) (R OIL_4_DIO.1) (R OIL_4_DIO.2) (R MILL_3_DIO.1) (R MILL_3_DIO.2) (R MILL_4_DIO.1) (R MILL_4_DIO.2) (R FAN_3_DIO.1) (R FAN_3_DIO.2) (R FAN_4_DIO.1) (R FAN_4_DIO.2) (R CONV_3_DIO.1) (R CONV_3_DIO.2) (R CONV_4_DIO.1) (R CONV_4_DIO.2) (R VIBR_3_DIO.1) (R VIBR_4_DIO.1) (R HORN_RUN_3) (S ELEV_0_DIO.11)
NETWORK 2
	{ [RESET_3] | [RESET_3] } - tpKVIT:TP(IN: *, PT: kvitVaqt)
_END_LD_
(* the same logic as Structured Text *)
(* Network 1 *)
_p1 := RESET_3 OR RESET_4 OR MILL_3.2 OR MILL_4.2 OR NOT ELEV_0_DIO.14;
IF _p1 THEN HORN_34_DIO.0 := TRUE; MILL_4.2 := FALSE; MILL_3.2 := FALSE; ELEV_34_DIO.1 := FALSE; ELEV_34_DIO.2 := FALSE; SHNEK_3_DIO.1 := FALSE; SHNEK_3_DIO.2 := FALSE; SHNEK_4_DIO.1 := FALSE; SHNEK_4_DIO.2 := FALSE; SHNK_SIKL_3_DIO.1 := FALSE; SHNK_SIKL_3_DIO.2 := FALSE; SHNK_SIKL_4_DIO.1 := FALSE; SHNK_SIKL_4_DIO.2 := FALSE; STAR_31_DIO.1 := FALSE; STAR_31_DIO.2 := FALSE; STAR_32_DIO.1 := FALSE; STAR_32_DIO.2 := FALSE; STAR_41_DIO.1 := FALSE; STAR_41_DIO.2 := FALSE; STAR_42_DIO.1 := FALSE; STAR_42_DIO.2 := FALSE; SEP_3_DIO.1 := FALSE; SEP_3_DIO.2 := FALSE; SEP_4_DIO.1 := FALSE; SEP_4_DIO.2 := FALSE; OIL_3_DIO.1 := FALSE; OIL_3_DIO.2 := FALSE; OIL_4_DIO.1 := FALSE; OIL_4_DIO.2 := FALSE; MILL_3_DIO.1 := FALSE; MILL_3_DIO.2 := FALSE; MILL_4_DIO.1 := FALSE; MILL_4_DIO.2 := FALSE; FAN_3_DIO.1 := FALSE; FAN_3_DIO.2 := FALSE; FAN_4_DIO.1 := FALSE; FAN_4_DIO.2 := FALSE; CONV_3_DIO.1 := FALSE; CONV_3_DIO.2 := FALSE; CONV_4_DIO.1 := FALSE; CONV_4_DIO.2 := FALSE; VIBR_3_DIO.1 := FALSE; VIBR_4_DIO.1 := FALSE; HORN_RUN_3 := FALSE; ELEV_0_DIO.11 := TRUE; END_IF;
(* Network 2 *)
tpKVIT(IN := RESET_3 OR RESET_3, PT := kvitVaqt);
END_PROGRAM

(* POU TRANSLATE, ST *)
PROGRAM TRANSLATE
VAR
	CON1: A_CONVER;
	CON2: A_CONVER;
	CON3: MY_LIN_TRAFO;
	CON4: A_CONVER;
	CON5: MY_LIN_TRAFO;
	CON6: A_CONVER;
	CON7: A_CONVER;
	CON8: A_CONVER;
	IN_MIN : REAL := 4;
	IN_MAX: REAL := 20;
	OUT_MIN_SEN : REAL := -10;
	OUT_MAX_SEN: REAL := 1;
	OUT_MIN_CUR : REAL := 0;
	OUT_MAX_CUR: REAL := 50;

	ELEV_34_CURRENT_4545: REAL;
	SHNEK_3_CURRENT_4545: REAL;
	FAN_4_SUCTION_41121: REAL;
	SHNEK_4_CURRENT_111: REAL;
	FAN_3_SUCTION_7777: REAL;
	ELEV_0_CURRENT_45465: REAL;
	SHOK_2_CURRENT_555: REAL;
	SHOK_1_CURRENT_4444: REAL;
END_VAR
freqTask();


MV8();
MV16();
MV24();
MU32_OUT();
MV48();
TANK_34_DIO.0 := TANK_MIN;
TANK_34_DIO.1 := TANK_MIDL;
TANK_34_DIO.2 := TANK_MAX;
hour_MOVE();
workHour();
ovn();
END_PROGRAM
ACTION hour_MOVE:
CONV_3_stopTIME := CONV_3_stopTIME_W;
CONV_3_startTIME := CONV_3_startTIME_W;
FAN_3_stopTIME := FAN_3_stopTIME_W;
FAN_3_startTIME := FAN_3_startTIME_W;
MILL_3_stopTIME := MILL_3_stopTIME_W;
MILL_3_startTIME := MILL_3_startTIME_W;
SEP_3_stopTIME := SEP_3_stopTIME_W;
SEP_3_startTIME := SEP_3_startTIME_W;
CONV_4_stopTIME := CONV_4_stopTIME_W;
CONV_4_startTIME := CONV_4_startTIME_W;
FAN_4_stopTIME := FAN_4_stopTIME_W;
FAN_4_startTIME := FAN_4_startTIME_W;
MILL_4_stopTIME := MILL_4_stopTIME_W;
MILL_4_startTIME := MILL_4_startTIME_W;
SEP_4_stopTIME := SEP_4_stopTIME_W;
SEP_4_startTIME:= SEP_4_startTIME_W;
ELEV_34_stopTIME := ELEV_34_stopTIME_W;
ELEV_34_startTIME := ELEV_34_startTIME_W;
SHNEK_3_stopTIME := SHNEK_3_stopTIME_W;
SHNEK_4_stopTIME := SHNEK_4_stopTIME_W;
SHNEK_3_startTIME := SHNEK_3_startTIME_W;
SHNEK_4_startTIME := SHNEK_4_startTIME_W;
STAR_31_stopTIME := STAR_31_stopTIME_W;
STAR_31_startTIME := STAR_31_startTIME_W;
STAR_32_stopTIME := STAR_32_stopTIME_W;
STAR_32_startTIME := STAR_32_startTIME_W;
STAR_41_stopTIME := STAR_41_stopTIME_W;
STAR_41_startTIME := STAR_41_startTIME_W;
STAR_42_stopTIME := STAR_42_stopTIME_W;
STAR_42_startTIME := STAR_42_startTIME_W;
OIL_3_stopTIME := OIL_3_stopTIME_W;
OIL_3_startTIME := OIL_3_startTIME_W;
OIL_4_stopTIME := OIL_4_stopTIME_W;
OIL_4_startTIME := OIL_4_startTIME_W;
SHNK_SIKL_3_stopTIME := SHNK_SIKL_3_stopTIME_W;
SHNK_SIKL_3_startTIME := SHNK_SIKL_3_startTIME_W;
SHNK_SIKL_4_stopTIME := SHNK_SIKL_4_stopTIME_W;
SHNK_SIKL_4_startTIME := SHNK_SIKL_4_startTIME_W;
END_ACTION
ACTION MB_ANALOG2:
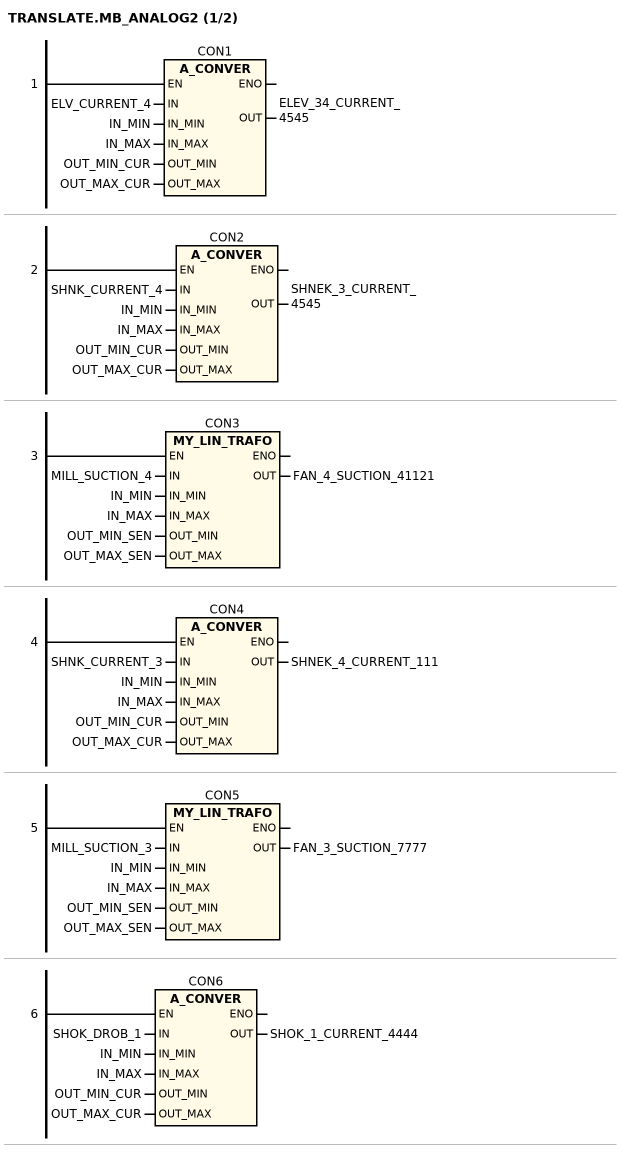
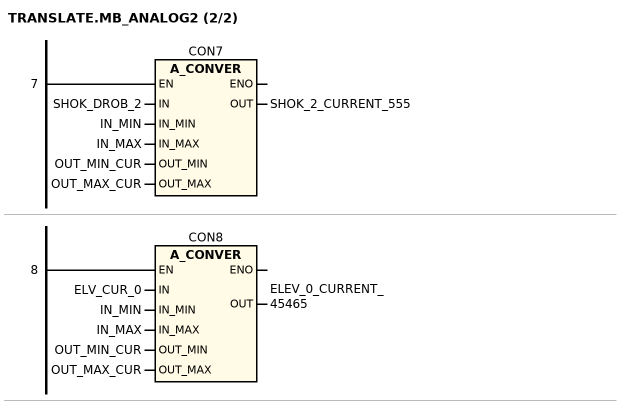
_LD_ (* Ladder Diagram *)
NETWORK 1
	*
		EN --- CON1:A_CONVER(IN: ELV_CURRENT_4, IN_MIN: IN_MIN, IN_MAX: IN_MAX, OUT_MIN: OUT_MIN_CUR, OUT_MAX: OUT_MAX_CUR) => ELEV_34_CURRENT_4545
NETWORK 2
	*
		EN --- CON2:A_CONVER(IN: SHNK_CURRENT_4, IN_MIN: IN_MIN, IN_MAX: IN_MAX, OUT_MIN: OUT_MIN_CUR, OUT_MAX: OUT_MAX_CUR) => SHNEK_3_CURRENT_4545
NETWORK 3
	*
		EN --- CON3:MY_LIN_TRAFO(IN: MILL_SUCTION_4, IN_MIN: IN_MIN, IN_MAX: IN_MAX, OUT_MIN: OUT_MIN_SEN, OUT_MAX: OUT_MAX_SEN) => FAN_4_SUCTION_41121
NETWORK 4
	*
		EN --- CON4:A_CONVER(IN: SHNK_CURRENT_3, IN_MIN: IN_MIN, IN_MAX: IN_MAX, OUT_MIN: OUT_MIN_CUR, OUT_MAX: OUT_MAX_CUR) => SHNEK_4_CURRENT_111
NETWORK 5
	*
		EN --- CON5:MY_LIN_TRAFO(IN: MILL_SUCTION_3, IN_MIN: IN_MIN, IN_MAX: IN_MAX, OUT_MIN: OUT_MIN_SEN, OUT_MAX: OUT_MAX_SEN) => FAN_3_SUCTION_7777
NETWORK 6
	*
		EN --- CON6:A_CONVER(IN: SHOK_DROB_1, IN_MIN: IN_MIN, IN_MAX: IN_MAX, OUT_MIN: OUT_MIN_CUR, OUT_MAX: OUT_MAX_CUR) => SHOK_1_CURRENT_4444
NETWORK 7
	*
		EN --- CON7:A_CONVER(IN: SHOK_DROB_2, IN_MIN: IN_MIN, IN_MAX: IN_MAX, OUT_MIN: OUT_MIN_CUR, OUT_MAX: OUT_MAX_CUR) => SHOK_2_CURRENT_555
NETWORK 8
	*
		EN --- CON8:A_CONVER(IN: ELV_CUR_0, IN_MIN: IN_MIN, IN_MAX: IN_MAX, OUT_MIN: OUT_MIN_CUR, OUT_MAX: OUT_MAX_CUR) => ELEV_0_CURRENT_45465
_END_LD_
(* the same logic as Structured Text *)
(* Network 1 *)
CON1(IN := ELV_CURRENT_4, IN_MIN := IN_MIN, IN_MAX := IN_MAX, OUT_MIN := OUT_MIN_CUR, OUT_MAX := OUT_MAX_CUR);
ELEV_34_CURRENT_4545 := CON1.OUT;
(* Network 2 *)
CON2(IN := SHNK_CURRENT_4, IN_MIN := IN_MIN, IN_MAX := IN_MAX, OUT_MIN := OUT_MIN_CUR, OUT_MAX := OUT_MAX_CUR);
SHNEK_3_CURRENT_4545 := CON2.OUT;
(* Network 3 *)
CON3(IN := MILL_SUCTION_4, IN_MIN := IN_MIN, IN_MAX := IN_MAX, OUT_MIN := OUT_MIN_SEN, OUT_MAX := OUT_MAX_SEN);
FAN_4_SUCTION_41121 := CON3.OUT;
(* Network 4 *)
CON4(IN := SHNK_CURRENT_3, IN_MIN := IN_MIN, IN_MAX := IN_MAX, OUT_MIN := OUT_MIN_CUR, OUT_MAX := OUT_MAX_CUR);
SHNEK_4_CURRENT_111 := CON4.OUT;
(* Network 5 *)
CON5(IN := MILL_SUCTION_3, IN_MIN := IN_MIN, IN_MAX := IN_MAX, OUT_MIN := OUT_MIN_SEN, OUT_MAX := OUT_MAX_SEN);
FAN_3_SUCTION_7777 := CON5.OUT;
(* Network 6 *)
CON6(IN := SHOK_DROB_1, IN_MIN := IN_MIN, IN_MAX := IN_MAX, OUT_MIN := OUT_MIN_CUR, OUT_MAX := OUT_MAX_CUR);
SHOK_1_CURRENT_4444 := CON6.OUT;
(* Network 7 *)
CON7(IN := SHOK_DROB_2, IN_MIN := IN_MIN, IN_MAX := IN_MAX, OUT_MIN := OUT_MIN_CUR, OUT_MAX := OUT_MAX_CUR);
SHOK_2_CURRENT_555 := CON7.OUT;
(* Network 8 *)
CON8(IN := ELV_CUR_0, IN_MIN := IN_MIN, IN_MAX := IN_MAX, OUT_MIN := OUT_MIN_CUR, OUT_MAX := OUT_MAX_CUR);
ELEV_0_CURRENT_45465 := CON8.OUT;
END_ACTION
ACTION MU32_OUT:
MU01 := BOOL_TO_WORD(ELV_RUN) * 1000;
MU02 := BOOL_TO_WORD(SHNK_RUN_4) * 1000;
MU03 := BOOL_TO_WORD(SHNK_SKL_RUN_4) * 1000;
MU04 := BOOL_TO_WORD(STAR_RUN_41) * 1000;
MU05 := BOOL_TO_WORD(STAR_RUN_42) * 1000;
MU06 := BOOL_TO_WORD(SEPR_RUN_4) * 1000;
MU07 := BOOL_TO_WORD(OIL_ST_RUN_4) * 1000;
MU08 := BOOL_TO_WORD(MILL_RUN_4) * 1000;
MU09 := BOOL_TO_WORD(FAN_RUN_4) * 1000;
MU10 := BOOL_TO_WORD(CONV_RUN_4) * 1000;
MU11 := BOOL_TO_WORD(VIBR_RUN_4) * 1000;
MU12 := BOOL_TO_WORD(VALV_RUN_4) * 1000;
MU13 := BOOL_TO_WORD(HORN_RUN_4) * 1000;
(*
MU14 := BOOL_TO_WORD(m_out14) * 1000;
MU15 := BOOL_TO_WORD(m_out15) * 1000;
MU16 := BOOL_TO_WORD(m_out16) * 1000;
*)
MU17 := BOOL_TO_WORD(ELV_RUN) * 1000;
MU18 := BOOL_TO_WORD(SHNK_RUN_3) * 1000;
MU19 := BOOL_TO_WORD(SHNK_SKL_RUN_3) * 1000;
MU20 := BOOL_TO_WORD(STAR_RUN_31) * 1000;
MU21 := BOOL_TO_WORD(STAR_RUN_32) * 1000;
MU22 := BOOL_TO_WORD(SEPR_RUN_3) * 1000;
MU23 := BOOL_TO_WORD(OIL_ST_RUN_3) * 1000;
MU24 := BOOL_TO_WORD(MILL_RUN_3) * 1000;
MU25 := BOOL_TO_WORD(FAN_RUN_3) * 1000;
MU26 := BOOL_TO_WORD(CONV_RUN_3) * 1000;
MU27 := BOOL_TO_WORD(VIBR_RUN_3) * 1000;
MU28 := BOOL_TO_WORD(VALV_RUN_3) * 1000;
MU29 := BOOL_TO_WORD(HORN_RUN_3) * 1000;
(*
MU30 := BOOL_TO_WORD(m_out30) * 1000;
MU31 := BOOL_TO_WORD(m_out31) * 1000;
MU32 := BOOL_TO_WORD(m_out32) * 1000;
*)
END_ACTION
ACTION MV16:
STAR_STOP_32 := MV16_0.0;
SEPR_STOP_3 := MV16_0.1;
OIL_ST_STOP_3 := MV16_0.2;
MILL_STOP_3 := MV16_0.3;
FAN_STOP_3 := MV16_0.4;
CONV_STOP_3 := MV16_0.5;
VIBR_STOP_3 := MV16_0.6;
(**********************)

STAR_START_32 := MV16_0.8;
SEPR_START_3 := MV16_0.9;
OIL_ST_START_3 := MV16_0.10;
MILL_START_3 := MV16_0.11;
FAN_START_3 := MV16_0.12;
CONV_START_3 := MV16_0.13;
VIBR_START_3 := MV16_0.14;
END_ACTION
ACTION MV24:
ELV_KM := MV24_0.0;
SHNK_KM_4 := MV24_0.1;
SHNK_SKL_KM_4 := MV24_0.2;
STAR_KM_41 := MV24_0.3;
STAR_KM_42 := MV24_0.4;
SEPR_KM_4 := MV24_0.5;
OIL_ST_KM_4 := MV24_0.6;
MILL_KM_4 := MV24_0.7;
MILL_4_DIO.8 := MATER_FULL_4 := MV24_0.8;
FAN_KM_4 := MV24_0.9;
CONV_KM_4 := MV24_0.10;
VIBR_KM_4 := MV24_0.11;
(*********
ELV_KM_3 := MV24_1.0;*)
SHNK_KM_3 := MV24_1.1;
SHNK_SKL_KM_3 := MV24_1.2;
STAR_KM_31 := MV24_1.3;
STAR_KM_32 := MV24_1.4;
SEPR_KM_3 := MV24_1.5;
OIL_ST_KM_3 := MV24_1.6;
MILL_KM_3 := MV24_1.7;
MILL_3_DIO.8 := MATER_FULL_3 := MV24_1.8;
FAN_KM_3 := MV24_1.9;
CONV_KM_3 := MV24_1.10;
VIBR_KM_3 := MV24_1.11;
CONTR_PHASE_1_2  := MV24_1.12;
END_ACTION
ACTION MV48:
	EMER_STOP_0 := MV48_0.0;
	MANUAL_ELV_0 := MV48_0.1;
	AUTO_ELV_0 := MV48_0.2;
	RESET_0 := MV48_0.3;
	ELV_STOP_0 := MV48_0.4;
	ELV_START_0 := MV48_0.5;
	SHOK_DROB_STOP_1  := MV48_0.6;
	SHOK_DROB_START_1 := MV48_0.7;
	SHOK_DROB_STOP_2  := MV48_0.8;
	SHOK_DROB_START_2 := MV48_0.9;
	CONV_STOP_0 := MV48_0.10;
	CONV_START_0 := MV48_0.11;
	(****RESERV CONV ***) (*12*)
	(***RESERV CONV****) (*13*)
	ELV_KM_0 := MV48_0.14;
	SHOK_DROB_KM_1 := MV48_0.15;
	SHOK_DROB_KM_2 := MV48_1.0;
	CONV_KM_0 := MV48_1.1;
	(** RESERV KM CONV **)
	TANK_MAX_0 := MV48_1.3;
	TANK_MIDLE_0 := MV48_1.4;
	TANK_MIN_0 := MV48_1.5;
END_ACTION
ACTION MV8:
ELV_STOP_4 := MV8_0.0;
SHNK_STOP_4 := MV8_0.1;
SHNK_SKL_STOP_4 := MV8_0.2;
STAR_STOP_41 := MV8_0.3;
STAR_STOP_42 := MV8_0.4;
SEPR_STOP_4 := MV8_0.5;
OIL_ST_STOP_4 := MV8_0.6;
MILL_STOP_4 := MV8_0.7;
FAN_STOP_4 := MV8_0.8;
CONV_STOP_4 := MV8_0.9;
VIBR_STOP_4 := MV8_0.10;

ELV_STOP_3 := MV8_0.12;
SHNK_STOP_3 := MV8_0.13;
SHNK_SKL_STOP_3 := MV8_0.14;
STAR_STOP_31 := MV8_0.15;

(**********************)
ELV_START_4 := MV8_1.0;
SHNK_START_4 := MV8_1.1;
SHNK_SKL_START_4 := MV8_1.2;
STAR_START_41 := MV8_1.3;
STAR_START_42 := MV8_1.4;
SEPR_START_4 := MV8_1.5;
OIL_ST_START_4 := MV8_1.6;
MILL_START_4 := MV8_1.7;
FAN_START_4 := MV8_1.8;
CONV_START_4 := MV8_1.9;
VIBR_START_4 := MV8_1.10;

ELV_START_3 := MV8_1.12;
SHNK_START_3 := MV8_1.13;
SHNK_SKL_START_3 := MV8_1.14;
STAR_START_31 := MV8_1.15;
END_ACTION
ACTION ovn:
ELEV_34_CURRENT := ELV_CURRENT_4;
SHNEK_3_CURRENT := SHNK_CURRENT_4;
FAN_4_SUCTION := MILL_SUCTION_4;
SHNEK_4_CURRENT := SHNK_CURRENT_3;
FAN_3_SUCTION := MILL_SUCTION_3;

SHOK_1_CURRENT := SHOK_DROB_1;
SHOK_2_CURRENT := SHOK_DROB_2;
ELEV_0_CURRENT := ELV_CUR_0;
END_ACTION
ACTION TR_REG_1:
(*
REG_1.0 := MB_ELV_ALR;
REG_1.1 := MB_ELV_ALR_ENC;
REG_1.2 := MB_SHNK_ALR_4;
REG_1.3 :=MB_SHNK_ENC_ALR_4 ;
REG_1.4 := MB_SHNK_SKL_ALR_4;
REG_1.5 := MB_SHNK_SKL_ENC_ALR_4;
REG_1.6 :=MB_STAR_ALR_41 ;
REG_1.7 := MB_STAR_ALR_42;

REG_1.8 := MB_SEPR_ALR_4;
REG_1.9 := MB_OIL_ST_ALR_4;
REG_1.10 :=MB_MILL_ALR_4 ;
REG_1.11 := MB_FAN_ALR_4;
REG_1.12 := MB_CONV_ALR_4;
REG_1.13 := MB_VIBR_ALR_4 ;
REG_1.14 := MB_MILL_ENC_ALR_4;
REG_1.15 := MB_SEPR_ENC_ALR_4;
*);
END_ACTION
ACTION TR_REG_2:
(*
REG_2.0 := MB_SHNK_ALR_3;
REG_2.1 := MB_SHNK_ENC_ALR_3;
REG_2.2 := MB_SHNK_SKL_ALR_3;
REG_2.3 := MB_STAR_ALR_31;
REG_2.4 := MB_STAR_ALR_32;
REG_2.5 := MB_SEPR_ALR_3;
REG_2.6 := MB_SEPR_ENC_ALR_3;
REG_2.7 := MB_OIL_ST_ALR_3;

REG_2.8 := MB_MILL_ALR_3;
REG_2.10 := MB_FAN_ALR_3;
REG_2.11 := MB_CONV_ALR_3;
REG_2.12 := MB_VIBR_ALR_3;
REG_2.13 := MB_MILL_ENC_ALR_3;
REG_2.14 := MB_TANK_MIN;
REG_2.15 := MB_TANK_MAX;

*)
;
END_ACTION
ACTION TR_REG_3:
(*
REG_3.0 := MB_ELV_RUN;
REG_3.1 := MB_SHNK_RUN_4;
REG_3.2 := MB_SHNK_SKL_RUN_4;
REG_3.3 := MB_STAR_RUN_41;
REG_3.4 := MB_STAR_RUN_42;
REG_3.5 := MB_SEPR_RUN_4;
REG_3.6 := MB_OIL_ST_RUN_4;
REG_3.7 := MB_MILL_RUN_4;

REG_3.8 := MB_FAN_RUN_4;
REG_3.9 := MB_CONV_RUN_4;
REG_3.10 := MB_VIBR_RUN_4;
REG_3.11 := MB_VALV_RUN_4;
REG_3.12 := MB_HORN_RUN;
REG_3.13 := MB_MATER_FULL_4;

*)
;
END_ACTION
ACTION TR_REG_4:
(*
REG_4.0 := MB_SHNK_RUN_3;
REG_4.1 := MB_SHNK_SKL_RUN_3;
REG_4.2 := MB_STAR_RUN_31;
REG_4.3 := MB_STAR_RUN_32;
REG_4.4 := MB_SEPR_RUN_3;
REG_4.5 := MB_OIL_ST_RUN_3;
REG_4.6 := MB_MILL_RUN_3;
REG_4.7 := MB_FAN_RUN_3;

REG_4.8 := MB_CONV_RUN_3;
REG_4.9 := MB_VIBR_RUN_3;
REG_4.10 := MB_VALV_RUN_3;
REG_4.11 := MB_MATER_FULL_3;

*)
;
END_ACTION

(* POU A_CONVER, CFC *)
FUNCTION_BLOCK A_CONVER
VAR_INPUT
	IN : REAL;
	IN_MIN : REAL := 4;
	IN_MAX : REAL := 20;
	OUT_MIN : REAL := 4;
	OUT_MAX : REAL := 20;
END_VAR
VAR_OUTPUT
	OUT : INT;

END_VAR
VAR
	LIN1: LIN_TRAFO;
END_VAR
VAR (* helpers for the ST form of the networks *)
	_t11 : INT;
END_VAR
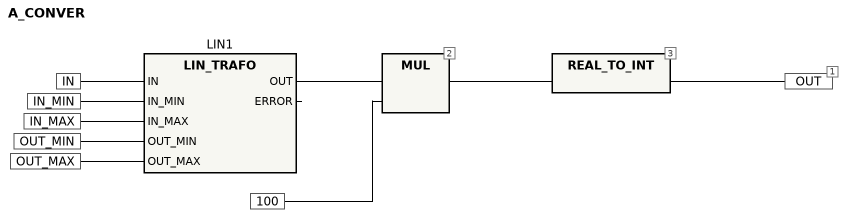
_CFC_ (* Continuous Function Chart, elements in execution order *)
#0 LIN1:LIN_TRAFO(IN: IN, IN_MIN: IN_MIN, IN_MAX: IN_MAX, OUT_MIN: OUT_MIN, OUT_MAX: OUT_MAX)
#1 OUT <= #3
#2 MUL(#0.OUT, 100)
#3 REAL_TO_INT(#2)
_END_CFC_
(* the same logic as Structured Text *)
LIN1(IN := IN, IN_MIN := IN_MIN, IN_MAX := IN_MAX, OUT_MIN := OUT_MIN, OUT_MAX := OUT_MAX);
OUT := _t11;
_t11 := REAL_TO_INT(LIN1.OUT * 100);
END_FUNCTION_BLOCK

(* POU MY_LIN_TRAFO, CFC *)
FUNCTION_BLOCK MY_LIN_TRAFO
VAR_INPUT
	IN : REAL;
	IN_MIN : REAL;
	IN_MAX : REAL;
	OUT_MIN : REAL;
	OUT_MAX : REAL;
END_VAR
VAR_OUTPUT
	OUT : REAL;
END_VAR
VAR
	TRA: LIN_TRAFO;
END_VAR
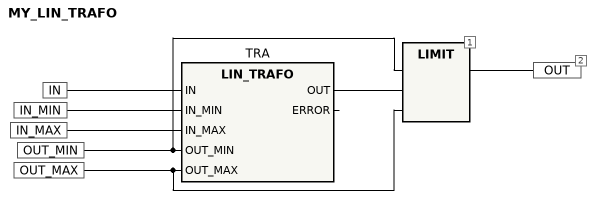
_CFC_ (* Continuous Function Chart, elements in execution order *)
#0 TRA:LIN_TRAFO(IN: IN, IN_MIN: IN_MIN, IN_MAX: IN_MAX, OUT_MIN: OUT_MIN, OUT_MAX: OUT_MAX)
#1 LIMIT(OUT_MIN, #0.OUT, OUT_MAX)
#2 OUT <= #1
_END_CFC_
(* the same logic as Structured Text *)
TRA(IN := IN, IN_MIN := IN_MIN, IN_MAX := IN_MAX, OUT_MIN := OUT_MIN, OUT_MAX := OUT_MAX);
OUT := LIMIT(OUT_MIN, TRA.OUT, OUT_MAX);
END_FUNCTION_BLOCK

(* POU freqTask, ST *)
PROGRAM freqTask
VAR
END_VAR
CONV_3_CURRENT := CONV_CURRENT_3;
CONV_3_FREQ := CONV_FREQ_3;
CONV_SET_FREQ_3 := CONV_3_SETPOINT;

FAN_3_CURRENT :=FAN_CURRENT_3;
FAN_3_FREQ := FAN_FREQ_3;
FAN_SET_FREQ_3 := FAN_3_SETPOINT;

MILL_3_CURRENT :=MILL_CURRENT_3;
MILL_3_FREQ := MILL_FREQ_3;
MILL_SET_FREQ_3 := MILL_3_SETPOINT;

SEP_3_CURRENT :=SEP_CURRENT_3;
SEP_3_FREQ := SEP_FREQ_3;
SEP_SET_FREQ_3 := SEP_3_SETPOINT;

CONV_4_CURRENT := CONV_CURRENT_4;
CONV_4_FREQ := CONV_FREQ_4;
CONV_SET_FREQ_4 := CONV_4_SETPOINT;

FAN_4_CURRENT :=FAN_CURRENT_4;
FAN_4_FREQ := FAN_FREQ_4;
FAN_SET_FREQ_4 := FAN_4_SETPOINT;

MILL_4_CURRENT :=MILL_CURRENT_4;
MILL_4_FREQ := MILL_FREQ_4;
MILL_SET_FREQ_4 := MILL_4_SETPOINT;

SEP_4_CURRENT :=SEP_CURRENT_4;
SEP_4_FREQ := SEP_FREQ_4;
SEP_SET_FREQ_4 := SEP_4_SETPOINT;



IF MILL_3.4 THEN
	CONV_PANEL_3 :=8;
	FAN_PANEL_3 :=9;
	MILL_PANEL_3 :=8;
	SEP_PANEL_3 :=8;
ELSE
	CONV_PANEL_3 :=0;
	FAN_PANEL_3 :=2;
	MILL_PANEL_3 :=0;
	SEP_PANEL_3 :=0;
END_IF;

IF MILL_4.4 THEN
	CONV_PANEL_4 :=8;
	FAN_PANEL_4 :=9;
	MILL_PANEL_4 :=8;
	SEP_PANEL_4 :=8;
ELSE
	CONV_PANEL_4 :=0;
	FAN_PANEL_4 :=2;
	MILL_PANEL_4 :=0;
	SEP_PANEL_4 :=0;
END_IF;
END_PROGRAM

(* POU workHour, LD *)
PROGRAM workHour
VAR
	evlev3_hour : calcHOUR;
	CONV_3_hour : calcHOUR;
	FAN_3_hour : calcHOUR;
	MILL_3_hour : calcHOUR;
	SEP_3_hour : calcHOUR;
	CONV_4_hour : calcHOUR;
	FAN_4_hour : calcHOUR;

	MILL_4_hour: calcHOUR;
	SEP_4_hour: calcHOUR;
	SHNEK_3_hour: calcHOUR;
	SHNEK_4_hour: calcHOUR;
	STAR_31_hour: calcHOUR;
	STAR_32_hour: calcHOUR;
	STAR_41_hour: calcHOUR;
	STAR_42_hour: calcHOUR;
	OIL_3_hour: calcHOUR;
	OIL_4_hour: calcHOUR;
	SHNK_SIKL_3_hour: calcHOUR;
	SHNK_SIKL_4_hour: calcHOUR;

	ELEV_0_hour: calcHOUR;
	SHOK_1_hour: calcHOUR;
	SHOK_2_hour: calcHOUR;
	CONV_0_hour: calcHOUR;
END_VAR
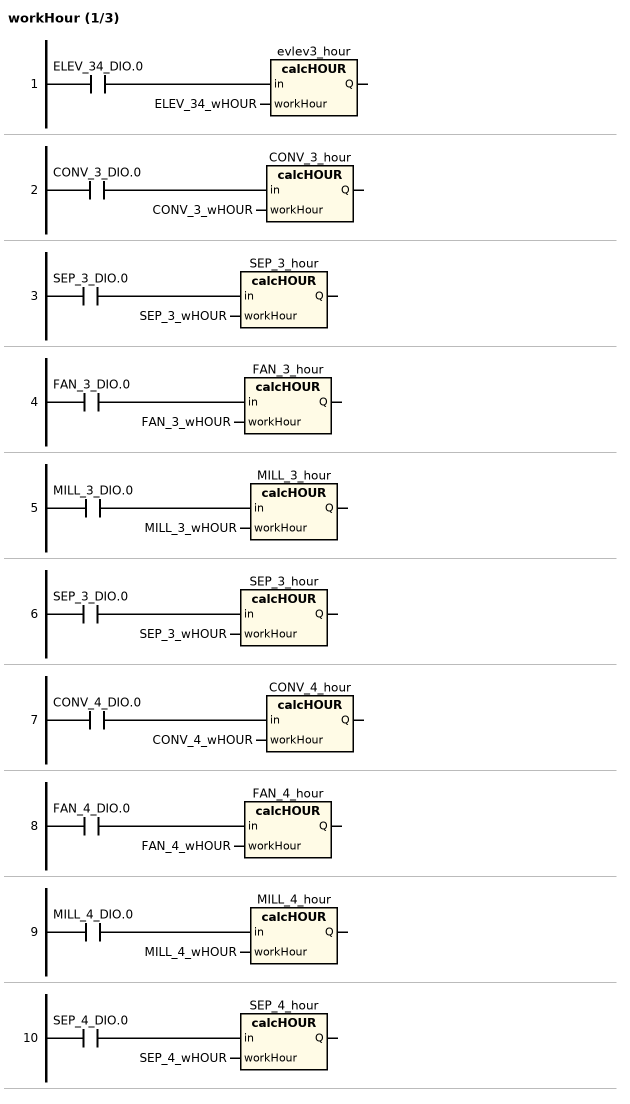
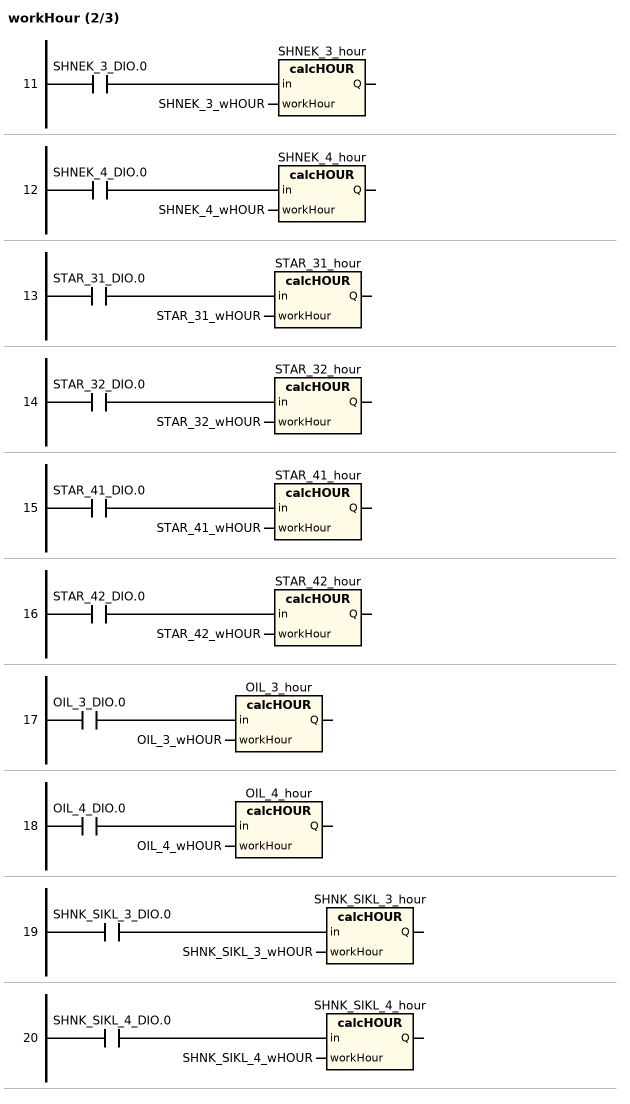
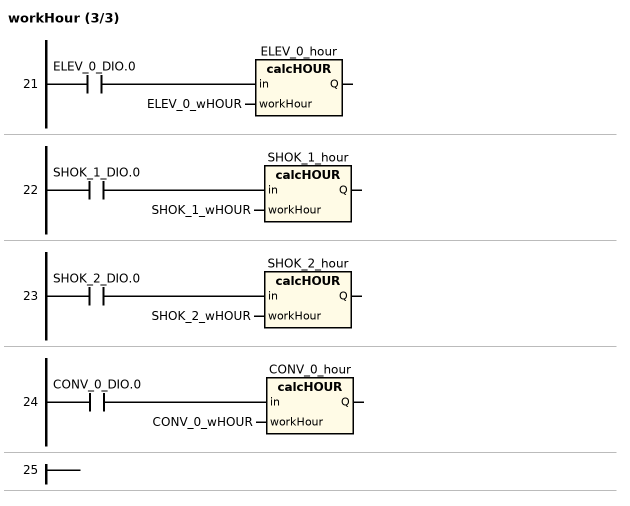
_LD_ (* Ladder Diagram *)
NETWORK 1
	[ELEV_34_DIO.0] - evlev3_hour:calcHOUR(in: *, workHour: ELEV_34_wHOUR)
NETWORK 2
	[CONV_3_DIO.0] - CONV_3_hour:calcHOUR(in: *, workHour: CONV_3_wHOUR)
NETWORK 3
	[SEP_3_DIO.0] - SEP_3_hour:calcHOUR(in: *, workHour: SEP_3_wHOUR)
NETWORK 4
	[FAN_3_DIO.0] - FAN_3_hour:calcHOUR(in: *, workHour: FAN_3_wHOUR)
NETWORK 5
	[MILL_3_DIO.0] - MILL_3_hour:calcHOUR(in: *, workHour: MILL_3_wHOUR)
NETWORK 6
	[SEP_3_DIO.0] - SEP_3_hour:calcHOUR(in: *, workHour: SEP_3_wHOUR)
NETWORK 7
	[CONV_4_DIO.0] - CONV_4_hour:calcHOUR(in: *, workHour: CONV_4_wHOUR)
NETWORK 8
	[FAN_4_DIO.0] - FAN_4_hour:calcHOUR(in: *, workHour: FAN_4_wHOUR)
NETWORK 9
	[MILL_4_DIO.0] - MILL_4_hour:calcHOUR(in: *, workHour: MILL_4_wHOUR)
NETWORK 10
	[SEP_4_DIO.0] - SEP_4_hour:calcHOUR(in: *, workHour: SEP_4_wHOUR)
NETWORK 11
	[SHNEK_3_DIO.0] - SHNEK_3_hour:calcHOUR(in: *, workHour: SHNEK_3_wHOUR)
NETWORK 12
	[SHNEK_4_DIO.0] - SHNEK_4_hour:calcHOUR(in: *, workHour: SHNEK_4_wHOUR)
NETWORK 13
	[STAR_31_DIO.0] - STAR_31_hour:calcHOUR(in: *, workHour: STAR_31_wHOUR)
NETWORK 14
	[STAR_32_DIO.0] - STAR_32_hour:calcHOUR(in: *, workHour: STAR_32_wHOUR)
NETWORK 15
	[STAR_41_DIO.0] - STAR_41_hour:calcHOUR(in: *, workHour: STAR_41_wHOUR)
NETWORK 16
	[STAR_42_DIO.0] - STAR_42_hour:calcHOUR(in: *, workHour: STAR_42_wHOUR)
NETWORK 17
	[OIL_3_DIO.0] - OIL_3_hour:calcHOUR(in: *, workHour: OIL_3_wHOUR)
NETWORK 18
	[OIL_4_DIO.0] - OIL_4_hour:calcHOUR(in: *, workHour: OIL_4_wHOUR)
NETWORK 19
	[SHNK_SIKL_3_DIO.0] - SHNK_SIKL_3_hour:calcHOUR(in: *, workHour: SHNK_SIKL_3_wHOUR)
NETWORK 20
	[SHNK_SIKL_4_DIO.0] - SHNK_SIKL_4_hour:calcHOUR(in: *, workHour: SHNK_SIKL_4_wHOUR)
NETWORK 21
	[ELEV_0_DIO.0] - ELEV_0_hour:calcHOUR(in: *, workHour: ELEV_0_wHOUR)
NETWORK 22
	[SHOK_1_DIO.0] - SHOK_1_hour:calcHOUR(in: *, workHour: SHOK_1_wHOUR)
NETWORK 23
	[SHOK_2_DIO.0] - SHOK_2_hour:calcHOUR(in: *, workHour: SHOK_2_wHOUR)
NETWORK 24
	[CONV_0_DIO.0] - CONV_0_hour:calcHOUR(in: *, workHour: CONV_0_wHOUR)
NETWORK 25
	*
_END_LD_
(* the same logic as Structured Text *)
(* Network 1 *)
evlev3_hour(in := ELEV_34_DIO.0, workHour := ELEV_34_wHOUR);
(* Network 2 *)
CONV_3_hour(in := CONV_3_DIO.0, workHour := CONV_3_wHOUR);
(* Network 3 *)
SEP_3_hour(in := SEP_3_DIO.0, workHour := SEP_3_wHOUR);
(* Network 4 *)
FAN_3_hour(in := FAN_3_DIO.0, workHour := FAN_3_wHOUR);
(* Network 5 *)
MILL_3_hour(in := MILL_3_DIO.0, workHour := MILL_3_wHOUR);
(* Network 6 *)
SEP_3_hour(in := SEP_3_DIO.0, workHour := SEP_3_wHOUR);
(* Network 7 *)
CONV_4_hour(in := CONV_4_DIO.0, workHour := CONV_4_wHOUR);
(* Network 8 *)
FAN_4_hour(in := FAN_4_DIO.0, workHour := FAN_4_wHOUR);
(* Network 9 *)
MILL_4_hour(in := MILL_4_DIO.0, workHour := MILL_4_wHOUR);
(* Network 10 *)
SEP_4_hour(in := SEP_4_DIO.0, workHour := SEP_4_wHOUR);
(* Network 11 *)
SHNEK_3_hour(in := SHNEK_3_DIO.0, workHour := SHNEK_3_wHOUR);
(* Network 12 *)
SHNEK_4_hour(in := SHNEK_4_DIO.0, workHour := SHNEK_4_wHOUR);
(* Network 13 *)
STAR_31_hour(in := STAR_31_DIO.0, workHour := STAR_31_wHOUR);
(* Network 14 *)
STAR_32_hour(in := STAR_32_DIO.0, workHour := STAR_32_wHOUR);
(* Network 15 *)
STAR_41_hour(in := STAR_41_DIO.0, workHour := STAR_41_wHOUR);
(* Network 16 *)
STAR_42_hour(in := STAR_42_DIO.0, workHour := STAR_42_wHOUR);
(* Network 17 *)
OIL_3_hour(in := OIL_3_DIO.0, workHour := OIL_3_wHOUR);
(* Network 18 *)
OIL_4_hour(in := OIL_4_DIO.0, workHour := OIL_4_wHOUR);
(* Network 19 *)
SHNK_SIKL_3_hour(in := SHNK_SIKL_3_DIO.0, workHour := SHNK_SIKL_3_wHOUR);
(* Network 20 *)
SHNK_SIKL_4_hour(in := SHNK_SIKL_4_DIO.0, workHour := SHNK_SIKL_4_wHOUR);
(* Network 21 *)
ELEV_0_hour(in := ELEV_0_DIO.0, workHour := ELEV_0_wHOUR);
(* Network 22 *)
SHOK_1_hour(in := SHOK_1_DIO.0, workHour := SHOK_1_wHOUR);
(* Network 23 *)
SHOK_2_hour(in := SHOK_2_DIO.0, workHour := SHOK_2_wHOUR);
(* Network 24 *)
CONV_0_hour(in := CONV_0_DIO.0, workHour := CONV_0_wHOUR);
(* Network 25 *)
END_PROGRAM

(* POU calcHOUR, CFC *)
FUNCTION_BLOCK calcHOUR
VAR_INPUT
	in : BOOL;
END_VAR
VAR_IN_OUT
	workHour : WORD;
END_VAR
VAR
	tp1: TP;
	go : BOOL;
	rtrig: R_TRIG;
	ctu1: CTU;
	vaqt : WORD := 3600;
END_VAR
VAR (* helpers for the ST form of the networks *)
	_t14 : WORD;
	_en14 : BOOL;
END_VAR
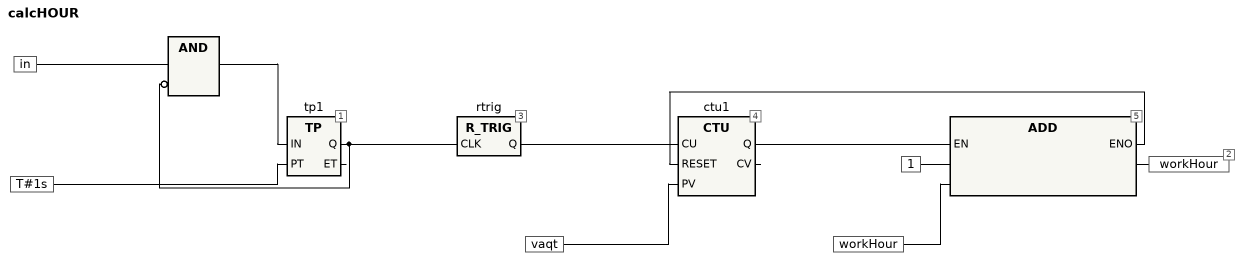
_CFC_ (* Continuous Function Chart, elements in execution order *)
#0 AND(in, NOT #1.Q)
#1 tp1:TP(IN: #0, PT: T#1s)
#2 workHour <= #5
#3 rtrig:R_TRIG(CLK: #1.Q)
#4 ctu1:CTU(CU: #3.Q, RESET: #5.ENO, PV: vaqt)
#5 ADD(EN: #4.Q, 1, workHour)
_END_CFC_
(* the same logic as Structured Text *)
tp1(IN := in AND NOT tp1.Q, PT := T#1s);
workHour := _t14;
rtrig(CLK := tp1.Q);
ctu1(CU := rtrig.Q, RESET := _en14, PV := vaqt);
_en14 := ctu1.Q;
IF _en14 THEN _t14 := 1 + workHour; END_IF;
END_FUNCTION_BLOCK

(* POU DROBILKA, LD *)
PROGRAM DROBILKA
VAR
	convTON : TON;
	conVAQT : TIME := T#180s;
	drobTON : TON;
	drobVAQT: TIME := T#180s;
	maxTON : TON;
	maxVAQT: TIME := T#5s;
	ELV_F_TRIG: F_TRIG;
	TANK_FULL: BOOL;
	ELV_R_TRIG: R_TRIG;
	vaqtInduc : WORD := 15;
	EL_0: ELEV_DR;
END_VAR
VAR (* helpers for the ST form of the networks *)
	_p1 : BOOL;
END_VAR
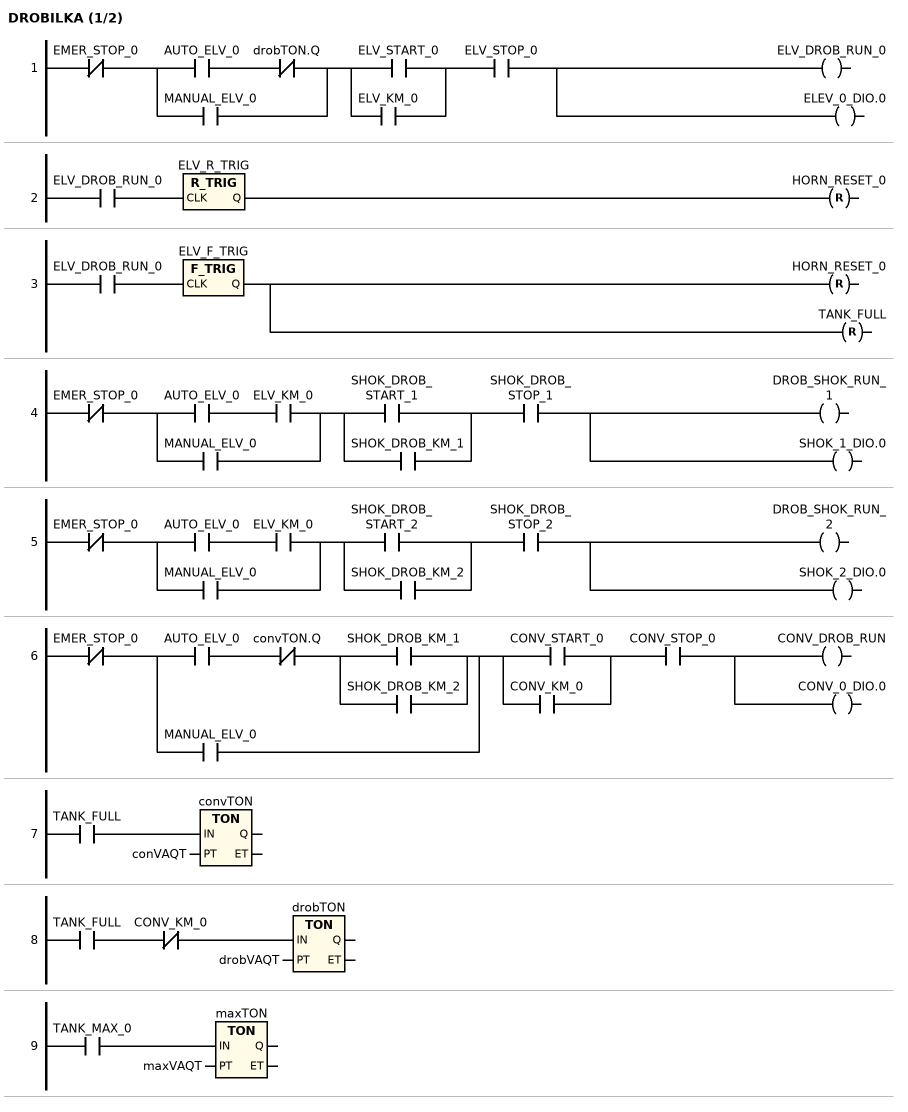
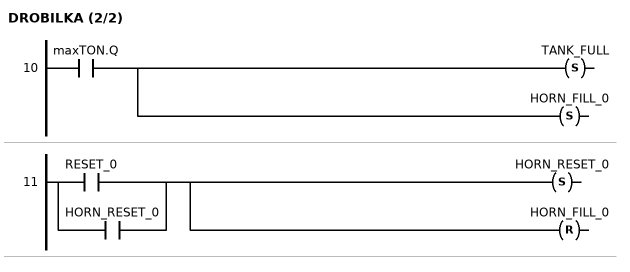
_LD_ (* Ladder Diagram *)
NETWORK 1
	[/EMER_STOP_0] - { [AUTO_ELV_0] - [/drobTON.Q] | [MANUAL_ELV_0] } - { [ELV_START_0] | [ELV_KM_0] } - [ELV_STOP_0] --- (ELV_DROB_RUN_0) (ELEV_0_DIO.0)
NETWORK 2
	[ELV_DROB_RUN_0] - ELV_R_TRIG:R_TRIG(CLK: *) --- (R HORN_RESET_0)
NETWORK 3
	[ELV_DROB_RUN_0] - ELV_F_TRIG:F_TRIG(CLK: *) --- (R HORN_RESET_0) (R TANK_FULL)
NETWORK 4
	[/EMER_STOP_0] - { [AUTO_ELV_0] - [ELV_KM_0] | [MANUAL_ELV_0] } - { [SHOK_DROB_START_1] | [SHOK_DROB_KM_1] } - [SHOK_DROB_STOP_1] --- (DROB_SHOK_RUN_1) (SHOK_1_DIO.0)
NETWORK 5
	[/EMER_STOP_0] - { [AUTO_ELV_0] - [ELV_KM_0] | [MANUAL_ELV_0] } - { [SHOK_DROB_START_2] | [SHOK_DROB_KM_2] } - [SHOK_DROB_STOP_2] --- (DROB_SHOK_RUN_2) (SHOK_2_DIO.0)
NETWORK 6
	[/EMER_STOP_0] - { [AUTO_ELV_0] - [/convTON.Q] - { [SHOK_DROB_KM_1] | [SHOK_DROB_KM_2] } | [MANUAL_ELV_0] } - { [CONV_START_0] | [CONV_KM_0] } - [CONV_STOP_0] --- (CONV_DROB_RUN) (CONV_0_DIO.0)
NETWORK 7
	[TANK_FULL] - convTON:TON(IN: *, PT: conVAQT)
NETWORK 8
	[TANK_FULL] - [/CONV_KM_0] - drobTON:TON(IN: *, PT: drobVAQT)
NETWORK 9
	[TANK_MAX_0] - maxTON:TON(IN: *, PT: maxVAQT)
NETWORK 10
	[maxTON.Q] --- (S TANK_FULL) (S HORN_FILL_0)
NETWORK 11
	{ [RESET_0] | [HORN_RESET_0] } --- (S HORN_RESET_0) (R HORN_FILL_0)
_END_LD_
(* the same logic as Structured Text *)
(* Network 1 *)
ELV_DROB_RUN_0 := NOT EMER_STOP_0 AND (AUTO_ELV_0 AND NOT drobTON.Q OR MANUAL_ELV_0) AND (ELV_START_0 OR ELV_KM_0) AND ELV_STOP_0;
ELEV_0_DIO.0 := ELV_DROB_RUN_0;
(* Network 2 *)
ELV_R_TRIG(CLK := ELV_DROB_RUN_0);
IF ELV_R_TRIG.Q THEN HORN_RESET_0 := FALSE; END_IF;
(* Network 3 *)
ELV_F_TRIG(CLK := ELV_DROB_RUN_0);
IF ELV_F_TRIG.Q THEN HORN_RESET_0 := FALSE; TANK_FULL := FALSE; END_IF;
(* Network 4 *)
DROB_SHOK_RUN_1 := NOT EMER_STOP_0 AND (AUTO_ELV_0 AND ELV_KM_0 OR MANUAL_ELV_0) AND (SHOK_DROB_START_1 OR SHOK_DROB_KM_1) AND SHOK_DROB_STOP_1;
SHOK_1_DIO.0 := DROB_SHOK_RUN_1;
(* Network 5 *)
DROB_SHOK_RUN_2 := NOT EMER_STOP_0 AND (AUTO_ELV_0 AND ELV_KM_0 OR MANUAL_ELV_0) AND (SHOK_DROB_START_2 OR SHOK_DROB_KM_2) AND SHOK_DROB_STOP_2;
SHOK_2_DIO.0 := DROB_SHOK_RUN_2;
(* Network 6 *)
CONV_DROB_RUN := NOT EMER_STOP_0 AND (AUTO_ELV_0 AND NOT convTON.Q AND (SHOK_DROB_KM_1 OR SHOK_DROB_KM_2) OR MANUAL_ELV_0) AND (CONV_START_0 OR CONV_KM_0) AND CONV_STOP_0;
CONV_0_DIO.0 := CONV_DROB_RUN;
(* Network 7 *)
convTON(IN := TANK_FULL, PT := conVAQT);
(* Network 8 *)
drobTON(IN := TANK_FULL AND NOT CONV_KM_0, PT := drobVAQT);
(* Network 9 *)
maxTON(IN := TANK_MAX_0, PT := maxVAQT);
(* Network 10 *)
IF maxTON.Q THEN TANK_FULL := TRUE; HORN_FILL_0 := TRUE; END_IF;
(* Network 11 *)
_p1 := RESET_0 OR HORN_RESET_0;
IF _p1 THEN HORN_RESET_0 := TRUE; HORN_FILL_0 := FALSE; END_IF;
END_PROGRAM

(* POU ELEV_DR, LD *)
FUNCTION_BLOCK ELEV_DR
VAR_INPUT (**********SHNEK *********)
	EN : BOOL;
	EMER_STOP_0: BOOL;
	EMER_STOP_0_VIRT : BOOL;
	AUTO_ELV_0 : BOOL;
	AUTO_ELV_VIRT : BOOL;
	MANUAL_ELV_0 : BOOL;
	ELV_START_0 : BOOL;
	ELV_START_0_VIRT : BOOL;

	ELV_START_0_ENC : BOOL;
	ELV_STOP_0 : BOOL;
	DROB_SHOK_RUN_2 : BOOL;
	DROB_SHOK_KM_ERROR : BOOL;
	SIMULATION : BOOL := TRUE;
	vaqtInduc : WORD := 15;
	ELEV_0_startTIME : WORD;
	ELEV_0_stopTIME : WORD;
END_VAR

VAR_OUTPUT
	OUT : BOOL;
	ALARM : BOOL;
END_VAR
VAR
	INDUK1: INDUKTIV;
	INDUK2: INDUKTIV;
	OUT_MAN: BOOL;
	OUT_AUTO: BOOL;
	START_TON : TON;
	STOP_TOF : TOF;
	startTIME : TIME;
	stopTIME : TIME;
	L1: BOOL;
	L2: BOOL;
	ES: BOOL;
	EMERGENCY_STOP: BOOL;
	ALARM1 : BOOL;
	ALARM2 : BOOL;

	STOP: BOOL;
	ALLOW: BOOL;
	START_timer: BOOL;
	STOP_timer: BOOL;
	TTT : TP;
END_VAR
VAR (* helpers for the ST form of the networks *)
	_p1 : BOOL;
END_VAR
